# B&R Automation Studio project TD52 (part 3)

## Logical view

Binary libraries used (declarations not repeated): AsString, AsTime, BrSystem, DataObj, FileIO, LoopConR 2.72.0, LoopCont 3.03.1, Operator, Runtime, standard, SYS_LIB, CAN_Lib, AsXml, AsIecCon, AsArLog, AsIO, AsIODiag, AsIOAcc, AsARCfg, DRV_mbus, dvframe, AsTCP, AsArProf, AsNxDpS, AsNxPnS, ModDiag 1.10.1, AsBrMath, ArEventLog, AsBrStr, AsIOVib, AsFltGen, ArFirewall, AsHW, AsANSL, MpBackup 5.24.2, MpBase 5.24.1, SfDomain 5.24.1, AsEPL, MpJ1939 5.24.2, lSAFI_VCD

### Package Logical/Libraries - Global Libraries

### Library Logical/Libraries/AmmBase (IEC, version 4.13.0) - +
Depends on: standard

#### AmmBase.typ - Exported data types
```iecst
TYPE
	MM2AmmBase : 	STRUCT
		bGnlTrip1 : BOOL;
		bGnlTrip2 : BOOL;
		bGnlTrip3 : BOOL;
		bTriptype1 : BOOL;
		bTriptype2 : BOOL;
		bTriptype3 : BOOL;
		bGnlWarning : BOOL;
		iMsg : ARRAY[0..9999]OF USINT;
	END_STRUCT;
	AmmBase2MM : 	STRUCT
		bResetTrip : BOOL;
		bResetWarning : BOOL;
		bGnlTrip1 : BOOL;
		bGnlTrip2 : BOOL;
		bGnlTrip3 : BOOL;
		bGnlWarning : BOOL;
		bResetRiskClass0 : BOOL;
		bResetRiskClass1 : BOOL;
		bResetRiskClass2 : BOOL;
		bResetRiskClass3 : BOOL;
		bResetRiskClass4 : BOOL;
		iNumAlmTest : UDINT;
	END_STRUCT;
END_TYPE
```

#### AmmBase.fun - Exported functions and function blocks
```iecst
FUNCTION_BLOCK Msg (*AMM*)
	VAR_INPUT
		Num : UINT; (*alarm number*)
		Enable : BOOL; (*alarm enable*)
		Set : BOOL; (*alarm set*)
		PT : TIME; (*alarm delay*)
		Prio : UINT; (*alarm priority*)
		RiskClass : UINT; (*alarm riskclass*)
		Reset : BOOL; (*alarm reset*)
		LockReset : BOOL; (*alarm reset locked out*)
		AmmInAdr : UDINT;
		AmmOutAdr : UDINT;
	END_VAR
	VAR_OUTPUT
		Q : BOOL;
		Status : UINT;
		Test : BOOL; (*alarm test active*)
	END_VAR
	VAR
		xSR : SR;
		xTON : TON;
		bAlmTest : BOOL;
		MM2AB : REFERENCE TO MM2AmmBase;
		AB2MM : REFERENCE TO AmmBase2MM;
		bAdressErr : BOOL;
	END_VAR
	VAR CONSTANT
		FUB_Msg_InAdr_Err : UINT := 1111;
		FUB_Msg_OutAdr_Err : UINT := 2222;
	END_VAR
	VAR
		bRemoteReset : BOOL;
		AsArLogWrite_AMM : AsArLogWrite;
		AsArLogGetInfo_0 : AsArLogGetInfo;
		SetLog : BOOL;
		zzEdge00000 : BOOL;
	END_VAR
END_FUNCTION_BLOCK
```

- AmmBase.st (not readable text: treated as protected, skipped)

### Library Logical/Libraries/JEW_LIB1 (ANSIC, version 1.93.0)
Depends on: brsystem, SYS_LIB, brsystem, SYS_LIB

#### JEW_LIB1.fun
```iecst
FUNCTION_BLOCK FILTER
	VAR_INPUT
		In : INT;
		Filter : USINT;
		Reset : BOOL;
	END_VAR
	VAR_OUTPUT
		Out : INT;
	END_VAR
	VAR
		temp_mw : DINT;
	END_VAR
END_FUNCTION_BLOCK

FUNCTION_BLOCK FILTER_R
	VAR_INPUT
		In : REAL;
		Filter : UINT;
		Reset : BOOL;
	END_VAR
	VAR_OUTPUT
		Out : REAL;
	END_VAR
	VAR
		temp_mw : LREAL;
	END_VAR
END_FUNCTION_BLOCK

FUNCTION_BLOCK TimeBasedOnOff
	VAR_INPUT
		enable : BOOL;
		x : INT;
		min_value : INT;
		max_value : INT;
		tchange : UDINT;
		hysteresis : UINT;
		set_pos : INT;
		basetime : UDINT;
	END_VAR
	VAR_OUTPUT
		down : BOOL;
		up : BOOL;
		y : INT;
		status : UINT;
	END_VAR
	VAR
		y_act : REAL;
		fHystUp : REAL;
		fHystDown : REAL;
		fUnitTime : REAL;
		ulLastTime : UDINT;
		fDiffTime : REAL;
		fHysteresis : REAL;
	END_VAR
END_FUNCTION_BLOCK

FUNCTION_BLOCK TimeBasedOnOff_R
	VAR_INPUT
		enable : BOOL;
		x : REAL;
		min_value : REAL;
		max_value : REAL;
		tchange : REAL;
		hysteresis : REAL;
		set_pos : REAL;
		basetime : REAL;
	END_VAR
	VAR_OUTPUT
		down : BOOL;
		up : BOOL;
		y : REAL;
		status : UINT;
	END_VAR
	VAR
		y_act : REAL;
		fHystUp : REAL;
		fHystDown : REAL;
		fUnitTime : REAL;
		ulLastTime : REAL;
		fDiffTime : REAL;
		fHysteresis : REAL;
	END_VAR
END_FUNCTION_BLOCK

FUNCTION_BLOCK WDtoBIT
	VAR_INPUT
		Word : UINT;
	END_VAR
	VAR_OUTPUT
		Bit00 : BOOL;
		Bit01 : BOOL;
		Bit02 : BOOL;
		Bit03 : BOOL;
		Bit04 : BOOL;
		Bit05 : BOOL;
		Bit06 : BOOL;
		Bit07 : BOOL;
		Bit08 : BOOL;
		Bit09 : BOOL;
		Bit10 : BOOL;
		Bit11 : BOOL;
		Bit12 : BOOL;
		Bit13 : BOOL;
		Bit14 : BOOL;
		Bit15 : BOOL;
	END_VAR
END_FUNCTION_BLOCK

FUNCTION_BLOCK BITtoWD
	VAR_INPUT
		Bit00 : BOOL;
		Bit01 : BOOL;
		Bit02 : BOOL;
		Bit03 : BOOL;
		Bit04 : BOOL;
		Bit05 : BOOL;
		Bit06 : BOOL;
		Bit07 : BOOL;
		Bit08 : BOOL;
		Bit09 : BOOL;
		Bit10 : BOOL;
		Bit11 : BOOL;
		Bit12 : BOOL;
		Bit13 : BOOL;
		Bit14 : BOOL;
		Bit15 : BOOL;
	END_VAR
	VAR_OUTPUT
		Word : UINT;
	END_VAR
END_FUNCTION_BLOCK

FUNCTION_BLOCK PID_A
	VAR_INPUT
		enable : BOOL;
		init : BOOL;
		ist : INT;
		soll : INT;
		kp : INT;
		ki : INT;
		kd : INT;
		gunten : INT;
		goben : INT;
		C0 : DINT;
	END_VAR
	VAR_OUTPUT
		limit : BOOL;
		integr : DINT;
		stell : INT;
	END_VAR
	VAR
		ist_alt : INT;
	END_VAR
END_FUNCTION_BLOCK

FUNCTION_BLOCK PID_A_R
	VAR_INPUT
		enable : BOOL;
		init : BOOL;
		ist : REAL;
		soll : REAL;
		kp : INT;
		ki : INT;
		kd : INT;
		gunten : INT;
		goben : INT;
		C0 : DINT;
	END_VAR
	VAR_OUTPUT
		limit : BOOL;
		integr : DINT;
		stell : REAL;
	END_VAR
	VAR
		ist_alt : INT;
	END_VAR
END_FUNCTION_BLOCK

FUNCTION_BLOCK TON_R
	VAR_INPUT
		IN : BOOL;
		PT : UDINT;
		RS : BOOL;
	END_VAR
	VAR_OUTPUT
		Q : BOOL;
		ET : UDINT;
	END_VAR
	VAR
		init_old : USINT;
		tick_old : UDINT;
	END_VAR
END_FUNCTION_BLOCK

FUNCTION_BLOCK BH
	VAR_INPUT
		enable : BOOL;
		BH_adr : UDINT;
	END_VAR
	VAR_OUTPUT
		BH_Imp : BOOL;
		BM_Imp : BOOL;
	END_VAR
END_FUNCTION_BLOCK

FUNCTION_BLOCK RAMPE
	VAR_INPUT
		enable : BOOL;
		In : INT;
		Rise : UINT;
		Sink : UINT;
		TC_Time : UINT;
	END_VAR
	VAR_OUTPUT
		Out : INT;
	END_VAR
	VAR
		f_out : REAL;
	END_VAR
END_FUNCTION_BLOCK

FUNCTION_BLOCK RAMPE_R
	VAR_INPUT
		enable : BOOL;
		In : REAL;
		Rise : REAL;
		Sink : REAL;
		TC_Time : UINT;
	END_VAR
	VAR_OUTPUT
		Out : REAL;
	END_VAR
	VAR
		f_out : REAL;
	END_VAR
END_FUNCTION_BLOCK

FUNCTION_BLOCK GR_MIN_MAXR
	VAR_INPUT
		In : REAL;
		Gw : REAL;
		Hy_min : REAL;
		Hy_max : REAL;
	END_VAR
	VAR_OUTPUT
		Q : BOOL;
	END_VAR
END_FUNCTION_BLOCK

FUNCTION_BLOCK GR_MIN
	VAR_INPUT
		In : INT;
		Gw : INT;
		Hy : INT;
	END_VAR
	VAR_OUTPUT
		Q : BOOL;
	END_VAR
END_FUNCTION_BLOCK

FUNCTION_BLOCK GR_MINR
	VAR_INPUT
		In : REAL;
		Gw : REAL;
		Hy : REAL;
	END_VAR
	VAR_OUTPUT
		Q : BOOL;
	END_VAR
END_FUNCTION_BLOCK

FUNCTION us_BitClr : UINT
	VAR_INPUT
		In : UINT;
		BitNr : USINT;
	END_VAR
END_FUNCTION

FUNCTION_BLOCK GR_MAX
	VAR_INPUT
		In : INT;
		Gw : INT;
		Hy : INT;
	END_VAR
	VAR_OUTPUT
		Q : BOOL;
	END_VAR
END_FUNCTION_BLOCK

FUNCTION_BLOCK GR_MAXR
	VAR_INPUT
		In : REAL;
		Gw : REAL;
		Hy : REAL;
	END_VAR
	VAR_OUTPUT
		Q : BOOL;
	END_VAR
END_FUNCTION_BLOCK

FUNCTION us_BitSet : UINT
	VAR_INPUT
		In : UINT;
		BitNr : USINT;
	END_VAR
END_FUNCTION

FUNCTION us_BitTest : BOOL
	VAR_INPUT
		In : UINT;
		BitNr : USINT;
	END_VAR
END_FUNCTION

FUNCTION uc_BitClr : USINT
	VAR_INPUT
		In : USINT;
		BitNr : USINT;
	END_VAR
END_FUNCTION

FUNCTION uc_BitSet : USINT
	VAR_INPUT
		In : USINT;
		BitNr : USINT;
	END_VAR
END_FUNCTION

FUNCTION uc_BitTest : BOOL
	VAR_INPUT
		In : USINT;
		BitNr : USINT;
	END_VAR
END_FUNCTION

FUNCTION ul_BitSet : UDINT
	VAR_INPUT
		In : UDINT;
		BitNr : USINT;
	END_VAR
END_FUNCTION

FUNCTION ul_BitClr : UDINT
	VAR_INPUT
		In : UDINT;
		BitNr : USINT;
	END_VAR
END_FUNCTION

FUNCTION ul_BitTest : BOOL
	VAR_INPUT
		In : UDINT;
		BitNr : USINT;
	END_VAR
END_FUNCTION

FUNCTION ITOA : SINT
	VAR_INPUT
		In : INT;
		Out : STRING[7];
	END_VAR
END_FUNCTION

FUNCTION_BLOCK xSignScal
	VAR_INPUT
		enable : BOOL;
		num : UINT;
		param : UDINT;
		In : INT;
	END_VAR
	VAR_OUTPUT
		error : BOOL;
		exceed : BOOL;
		Out : INT;
	END_VAR
END_FUNCTION_BLOCK

FUNCTION_BLOCK xSignScal_R
	VAR_INPUT
		enable : BOOL;
		num : UINT;
		param : UDINT;
		In : REAL;
	END_VAR
	VAR_OUTPUT
		error : BOOL;
		exceed : BOOL;
		Out : REAL;
	END_VAR
END_FUNCTION_BLOCK

FUNCTION_BLOCK TOF_R
	VAR_INPUT
		IN : BOOL;
		PT : UDINT;
		RS : BOOL;
	END_VAR
	VAR_OUTPUT
		Q : BOOL;
		ET : UDINT;
	END_VAR
	VAR
		init_old : UDINT;
		tick_old : UDINT;
	END_VAR
END_FUNCTION_BLOCK

FUNCTION_BLOCK TP_R
	VAR_INPUT
		IN : BOOL;
		PT : UDINT;
		RS : BOOL;
	END_VAR
	VAR_OUTPUT
		Q : BOOL;
		ET : UDINT;
	END_VAR
	VAR
		init_old : USINT;
		tick_old : UDINT;
		IN_old : BOOL;
	END_VAR
END_FUNCTION_BLOCK
```

#### JEW_LIB1.typ
```iecst
TYPE
	bh_typ : STRUCT
		tick	: USINT ;
		second	: USINT ;
		minute	: USINT ;
		spare	: USINT ;
	END_STRUCT;
END_TYPE
```

#### bh.c
```c
/***********************************************************************************
* Name      : bh.c
* Titel     : Betriebsstundengenerierung
* Version   : V1.10
* Datum     : 17.05.2002
*
* Uebergabe : enable			BOOL			Betriebsstundengenerierung aus/ein
*
* Rueckgabe : BH_adr	 struct USINT tick		Sekundentakt
*							    USINT second	Sekundenzaehler
*							    USINT minute	Minutenzähler
*								USINT spare		Reserve
*			  BH_Imp			BOOL			Betriebsstundenimpuls
*
* History   :
*  V1.00	  14.09.1998,fw			erstellt
*  V1.01	  24.08.2001,Fa.		fd->BD_adr durch fd->BH_adr ersetzt
*  V1.10	  17.05.2002,fw			#include <burtrap.h> durch <sys_lib.h> ersetzt
*  V1.70	  17.06.2002,WeitzerT	inc. plctypes entf.; bei jewlib1.h <> statt ""
*  V1.70.1	  24.01.2014,WeitzerT	correction of compiler warnings
*  V1.93.0	  27.10.2023,Zuschnig	Include minute impuls
*
***********************************************************************************/
#include <jew_lib1.h>
#include <sys_lib.h>

void BH(BH_typ *fd)
{
	UINT	ticks;
	bh_typ	*bh_adr;

	bh_adr = (bh_typ*)fd->BH_adr;

	fd->BH_Imp = 0;							/* vorab Stundenimpuls reset */
	fd->BM_Imp = 0;							/* vorab Minutenimpuls reset */

	if (fd->enable == 1)
	{
		ticks = 0;							/* Zwischenzeitlich für Änderung auf i386 */

		ticks = TIM_ticks();				/* 10 ms Takt auslesen */

		if ((ticks < 50) && (bh_adr->tick == 0))
		{
			bh_adr->tick = 1;				/* Sekundentakt setzen */
			++bh_adr->second;				/* im Sekundentakt zaehlen */
			if (bh_adr->second > 59)
			{
				bh_adr->second = 0;
				fd->BM_Imp = 1;				/* Minutenimpuls ausgeben */
				++bh_adr->minute;			/* im Minutetakt zaehlen */
				if (bh_adr->minute > 59)
				{
					fd->BH_Imp = 1;			/* Stundenimpuls ausgeben */
					bh_adr->minute = 0;
				}
			}
		}
		else if ((ticks > 50) && (bh_adr->tick == 1))
			bh_adr->tick = 0;				/* Sekundentakt ruecksetzen */
	}
}
```

#### bittowd.c
```c
/***********************************************************************************
* Name      : BITtoWD.c
* Titel     : 16 Bits auf ein Word(2Byte) komprimieren
* Version   : V1.00
* Datum     : 09.11.1998
*
* Uebergabe : Bit00		BOOL	Bit 00 des Ausgangswortes
*			  Bit01		BOOL	Bit 01 des Ausgangswortes
*			  Bit02		BOOL	Bit 02 des Ausgangswortes
*			  Bit03		BOOL	Bit 03 des Ausgangswortes
*			  Bit04		BOOL	Bit 04 des Ausgangswortes
*			  Bit05		BOOL	Bit 05 des Ausgangswortes
*			  Bit06		BOOL	Bit 06 des Ausgangswortes
*			  Bit07		BOOL	Bit 07 des Ausgangswortes
*			  Bit08		BOOL	Bit 08 des Ausgangswortes
*			  Bit09		BOOL	Bit 09 des Ausgangswortes
*			  Bit10		BOOL	Bit 10 des Ausgangswortes
*			  Bit11		BOOL	Bit 11 des Ausgangswortes
*			  Bit12		BOOL	Bit 12 des Ausgangswortes
*			  Bit13		BOOL	Bit 13 des Ausgangswortes
*			  Bit14		BOOL	Bit 14 des Ausgangswortes
*			  Bit15		BOOL	Bit 15 des Ausgangswortes
*
* Rueckgabe : Word 		UINT	Kompriemiertes Eingangsabbild
*
* History   :
*  V1.00	  09.11.1998,fw			erstellt
*  V1.70	  17.06.2002,WeitzerT	inc. plctypes entf.; bei jewlib1.h <> statt ""
*
***********************************************************************************/
#include <jew_lib1.h>

void BITtoWD(BITtoWD_typ *fd)
{
	fd->Word = fd->Bit15;
	fd->Word = ((fd->Word)<<1) + fd->Bit14;
	fd->Word = ((fd->Word)<<1) + fd->Bit13;
	fd->Word = ((fd->Word)<<1) + fd->Bit12;
	fd->Word = ((fd->Word)<<1) + fd->Bit11;
	fd->Word = ((fd->Word)<<1) + fd->Bit10;
	fd->Word = ((fd->Word)<<1) + fd->Bit09;
	fd->Word = ((fd->Word)<<1) + fd->Bit08;
	fd->Word = ((fd->Word)<<1) + fd->Bit07;
	fd->Word = ((fd->Word)<<1) + fd->Bit06;
	fd->Word = ((fd->Word)<<1) + fd->Bit05;
	fd->Word = ((fd->Word)<<1) + fd->Bit04;
	fd->Word = ((fd->Word)<<1) + fd->Bit03;
	fd->Word = ((fd->Word)<<1) + fd->Bit02;
	fd->Word = ((fd->Word)<<1) + fd->Bit01;
	fd->Word = ((fd->Word)<<1) + fd->Bit00;
}
```

#### filter.c
```c
/***********************************************************************************
* Name      : filter.c
* Titel     : Filter mit PT1-Verhalten
* Version   : V1.0
* Datum     : 14.09.1998
*
* Uebergabe : In		INT		Eingangssignal
*			  Filter	SINT	Filterkonstante filter = T1 / T (T1 = Verzoegerung 1. Ordnung)
*
* Rueckgabe : Out	 	INT		Ausgangssignal
*
* History   :
*  V1.00	  14.09.1998,fw		erstellt
*  V1.20      21.12.1998,BK		Zeitkonstante im .h-File von SINT auf USINT
*  V1.70	  17.06.2002,WeitzerT	inc. plctypes entf.; bei jewlib1.h <> statt ""
*  V1.91	  02.02.2022,Schmid		added Reset input
*
***********************************************************************************/
#include <jew_lib1.h>

void FILTER(FILTER_typ *fd)
{
	if (fd->Filter == 0)
		fd->Filter = 1;				/* Division durch 0 verhindern */

	if (fd->Reset)
		fd->temp_mw = fd->In * fd->Filter;
	else
		fd->temp_mw = fd->temp_mw + fd->In - fd->Out;

	fd->Out = (int)(fd->temp_mw/fd->Filter);
}
```

#### gr_max.c
```c
/***********************************************************************************
* Name      : gr_max.c
* Titel     : Maximal-Grenzwertkontrolle mit Hysterese
* Version   : V1.3
* Datum     : 28.09.1999
*
* Uebergabe : In		INT		Eingangssignal
*			  Gw		INT		Grenzwert
*			  Hy		INT		Hysterese
*
* Rueckgabe : Q	 		INT		Ausgangssignal = 1 => Grenzwert ueberschritten
*
* History   :
*  V1.00	  14.09.1998,fw			erstellt
*  V1.30      28.09.1999,BrunnerK	Vergleichsoperanden wurden geaendert
*  V1.70	  17.06.2002,WeitzerT	inc. plctypes entf.; bei jewlib1.h <> statt ""
*
***********************************************************************************/
#include <jew_lib1.h>

void GR_MAX(GR_MAX_typ *fd)
{
	if (fd->In >= fd->Gw)
		fd->Q = 1;
	else if (fd->In < (fd->Gw - fd->Hy))
		fd->Q = 0;
}
```

#### gr_min_maxR.c
```c
/***********************************************************************************
* Name      : gr_min_max.c
* Titel     : Maximal- and Minimum Grenzwertkontrolle mit Hysterese
* Version   : V1.3
* Datum     : 26.05.2015
*
* Uebergabe : In		INT		Eingangssignal
*			  Gw		INT		Grenzwert
*			  Hy_min	INT		Hysterese - Down limit
*			  Hy_max	INT		Hysterese - Up Limit
*
* Rueckgabe : Q	 		INT		Ausgangssignal = 1 => Grenzwert ueberschritten
*
* History   :
*  V1.00	  28.05.2015,Walid Mari  Erstellt, basiert auf GR_MAXR library
*
***********************************************************************************/
#include <jew_lib1.h>

void GR_MIN_MAXR(GR_MIN_MAXR_typ *fd)
{
	if 		(fd->In >=( fd->Gw	+	fd->Hy_max))
		fd->Q = 1;
	else if (fd->In < (fd->Gw 	- 	fd->Hy_min))
		fd->Q = 0;
}
```

#### gr_maxR.c
```c
/***********************************************************************************
* Name      : gr_max.c
* Titel     : Maximal-Grenzwertkontrolle mit Hysterese
* Version   : V1.3
* Datum     : 28.09.1999
*
* Uebergabe : In		INT		Eingangssignal
*			  Gw		INT		Grenzwert
*			  Hy		INT		Hysterese
*
* Rueckgabe : Q	 		INT		Ausgangssignal = 1 => Grenzwert ueberschritten
*
* History   :
*  V1.00	  14.09.1998,fw			erstellt
*  V1.30      28.09.1999,BrunnerK	Vergleichsoperanden wurden geaendert
*  V1.70	  17.06.2002,WeitzerT	inc. plctypes entf.; bei jewlib1.h <> statt ""
*
***********************************************************************************/
#include <jew_lib1.h>

void GR_MAXR(GR_MAXR_typ *fd)
{
	if (fd->In >= fd->Gw)
		fd->Q = 1;
	else if (fd->In < (fd->Gw - fd->Hy))
		fd->Q = 0;
}
```

#### gr_min.c
```c
/***********************************************************************************
* Name      : gr_min.c
* Titel     : Minimal-Grenzwertkontrolle mit Hysterese
* Version   : V1.3
* Datum     : 28.09.1999
*
* Uebergabe : In		INT		Eingangssignal
*			  Gw		INT		Grenzwert
*			  Hy		INT		Hysterese
*
* Rueckgabe : Q	 		INT		Ausgangssignal = 1 => Grenzwert unterschritten
*
* History   :
*  V1.00	  14.09.1998,fw			erstellt
*  V1.30      28.09.1999,BrunnerK	Vergleichsoperanden wurden geaendert
*  V1.70	  17.06.2002,WeitzerT	inc. plctypes entf.; bei jewlib1.h <> statt ""
*
***********************************************************************************/
#include <jew_lib1.h>

void GR_MIN(GR_MIN_typ *fd)
{
	if (fd->In <= fd->Gw)
		fd->Q = 1;
	else if (fd->In > (fd->Gw + fd->Hy))
		fd->Q = 0;
}
```

#### itoa.c
```c
/***********************************************************************************
* Name      : itoa.c
* Titel     : Konvertierung Integer to ASCII-String
* Version   : V1.3
* Datum     : 30.09.1999
*
* Uebergabe : Strukturvariable:
*             In		INT		Zu konvertierender Integerwert
*			  *pCharFld	SINT	Pointer auf das Char-Array
*
* Rueckgabe : Strukturvariable:
*			  StrLen	SINT	Laenge des Strings
*
* History   :
*  V1.00	  xx.xx.1998,fw			erstellt
*  V1.30      30.09.1999,BrunnerK	In Library umgewandelt
*  V1.70	  17.06.2002,WeitzerT	inc. plctypes entf.; bei jewlib1.h <> statt ""
*  V1.70.1	  24.01.2014,WeitzerT	correction of compiler warnings
*
***********************************************************************************/
#include <jew_lib1.h>

signed char ITOA(signed short In, plcstring* Out)

{
	signed short	i, string_len, neg;
	signed long		val;
	signed short	InTemp;

	string_len = 1;					/* minimum 1 Zeichen lang */
	neg = 0;						/* vorab Wert positiv */
	InTemp = 0;

	if (In<0)
	{								/* Wert negativ */
		InTemp = In;				/* Negative Wert sichern */
/*		In = abs(In);				   Absolutbetrag bilden */
		neg = 1;					/* Kennung Wert ist negativ setzen */
		string_len++;				/* String wird um das Vorzeichen länger */
		Out[0] = '-';		    	/* Vorzeichen am Stringanfang eintragen */
	}

	val = In;
	while((val= val/10) != 0)		/* Berechnung der Stringlänge */
	{
		string_len++;
	}

	val = In;
	Out[string_len] = 0;		/* Stringendekennung eintragen */

	for(i=0; i<(string_len-neg); ++i)	/* Wert ASCII wandeln */
	{
		Out[string_len-i-1] = (char)((val % 10) + '0');
		val = val / 10;
	}

	if (neg == 1)
	{
		In = InTemp;				/* Negativen Wert zuruecksichern */
	}

	return string_len;				/* Stringlänge ohne Stringendekennung */
}
```

#### pid_a_R.c
```c
/********************************************************************
 * COPYRIGHT -- INNIO Company
 ********************************************************************
 * Library: JEW_LIB1
 * File: pid_a_R.c
 * Author: 320003156
 * Created: August 17, 2011
 * Modified: 2017-08-08 FW   adapted for GCC 4.1.2.
 *******************************************************************/

#include <bur/plc.h>
#include <JEW_LIB1.h>

void PID_A_R(PID_A_R_typ* pida)
{
	/* Deklaration Zwischenablage */
	long	stell_neu;
	short	e;

	if (pida->enable)
	{
		/* Initialisierung Regler */
		if (pida->init)
		{
			pida->integr = pida->C0;
			pida->ist_alt = 0;
		}

		/* Rücksetzen von Limitfehler */
		pida->limit = 0;

		/* Regler - Algorythmus
		yi = yi_1 + (e + ist_alt)/2 * ki
		stell  = (yp + yi + yd) / 256
		stell  = (e*kp + yi + (ist_alt - e) * (kd * -1)) / 256
		*/

		/* Berechnung Regelabweichung */
		e = pida->soll - pida->ist;

		/* Berechnung Integralanteil */
		pida->integr = pida->integr + (pida->ki) * ((e + pida->ist_alt) >> 1);

		/* Berechnung Stellgröße */
		stell_neu = (pida->kp * e + pida->integr - pida->kd * (pida->ist_alt - e)) >> 8;

		/* Übergabe an Schnittstelle */
	    pida->stell = stell_neu;

		/* Prüfung und Begrenzung des Stellsignales */
        if (stell_neu < pida->gunten)
		{
			pida->limit = 1;
			if (pida->ki != 0) pida->integr = (pida->gunten << 8) - (pida->kp * e - pida->kd * (e - pida->ist_alt));
			pida->stell = pida->gunten;
		}
		else if (stell_neu > pida->goben)
		{
			pida->limit = 1;
			if (pida->ki != 0) pida->integr = (pida->goben << 8) - (pida->kp * e - pida->kd * (e - pida->ist_alt));
			pida->stell = pida->goben;
		}

		/* Übergabe für neue Berechnug */
		pida->ist_alt = e;

	}
}
```

#### pid_a.c
```c
/************************************************************************************
* Name      : pid_a.src                                                         	*
* Titel     : Einfacher PID-Regler auf Integer-Basis                               	*
*												                            	   	*
* Uebergabe : enable	BOOL	Freigabe											*
*			  init		BOOL	Initialisierung									   	*
*			  ist		INT		Inputvariablen, Istwert                         	*
*			  soll		INT		Sollwert                            	  			*
*			  kp		INT		Proportionalverstärkung                             *
*			  ki		INT		Integrationsbeiwert                                 *
*			  kd		INT		Differenzierbeiwert                                 *
*			  gunten	INT		unterer Grenzwert                              	   	*
*			  goben		INT		oberer Grenzwert                            	   	*
*			  C0		DINT	Integrator Startwert wird übernommen wenn !=0	   	*
*												                            	   	*
* Rueckgabe : limit		BOOL	Limit Stellgrenzwert unter-/Überschritten			*
*			  integr	DINT	Integrator              							*
*			  stell		INT		Outputvariable, Stellwert                           *
*												                       				*
* Lok. Var. : e			INT		Reglelabweichung aktuell							*
*			  ist_alt		INT		alte Regelabweichung für Differenzbildung			*
*			  stell_neu DINT	Zwischenspeicherung des Stellwertes					*
*												                            	   	*
* History   :	                            	   								   	*
* V1.00	  	  06.06.2002,tw		erstellt										   	*
* V1.10       2017-08-08 FW   adapted for GCC 4.1.2.
*																				   	*
*************************************************************************************
*               		                                                           	*
*  BESCHREIBUNG:        		                                                   	*
*  -------------                		                                           	*
*                                       		                                   	*
*  Der FUB PID_a realisiert einen einfachen PID-Algorithmus, der auf		       	*
*  unterschreiten der unteren Stellwertgrenze <gunten> und auf             		   	*
*  überschreiten der oberen Stellwertgrenze <goben> überwacht. In diesem		   	*
*  Fall wird der Integrator neu berechnet und der Stellwert gemäß der     		   	*
*  Grenze begrenzt.                                                       		   	*
*  Der Integrator <integr> muß beim erstmaligen Aufruf des FUB richtig    		   	*
*  initialisiert werden (in der Regel mit 0).                             		   	*
*  Die Regelparameter der FUB-Schnittstelle sind wegen der Integerrechnung		   	*
*  mit 256 zu multiplizieren, das untere Byte entspricht demnach der Stelle		   	*
*  hinter dem Komma.                                                      		   	*
*                                                                         		   	*
************************************************************************************/
#include <bur/plc.h>
#include <JEW_LIB1.h>

void PID_A(PID_A_typ* pida)
{
	/* Deklaration Zwischenablage */
	long	stell_neu;
	short	e;

	if (pida->enable)
	{
		/* Initialisierung Regler */
		if (pida->init)
		{
			pida->integr = pida->C0;
			pida->ist_alt = 0;
		}

		/* Rücksetzen von Limitfehler */
		pida->limit = 0;

		/* Regler - Algorythmus
		yi = yi_1 + (e + ist_alt)/2 * ki
		stell  = (yp + yi + yd) / 256
		stell  = (e*kp + yi + (ist_alt - e) * (kd * -1)) / 256
		*/

		/* Berechnung Regelabweichung */
		e = pida->soll - pida->ist;

		/* Berechnung Integralanteil */
		pida->integr = pida->integr + (pida->ki) * ((e + pida->ist_alt) >> 1);

		/* Berechnung Stellgröße */
		stell_neu = (pida->kp * e + pida->integr - pida->kd * (pida->ist_alt - e)) >> 8;

		/* Übergabe an Schnittstelle */
	    pida->stell = stell_neu;

		/* Prüfung und Begrenzung des Stellsignales */
        if (stell_neu < pida->gunten)
		{
			pida->limit = 1;
			if (pida->ki != 0) pida->integr = (pida->gunten << 8) - (pida->kp * e - pida->kd * (e - pida->ist_alt));
			pida->stell = pida->gunten;
		}
		else if (stell_neu > pida->goben)
		{
			pida->limit = 1;
			if (pida->ki != 0) pida->integr = (pida->goben << 8) - (pida->kp * e - pida->kd * (e - pida->ist_alt));
			pida->stell = pida->goben;
		}

		/* Übergabe für neue Berechnug */
		pida->ist_alt = e;

	}
}
```

#### rampe_R.c
```c
/********************************************************************
 * COPYRIGHT -- INNIO Company
 ********************************************************************
 * Library: JEW_LIB1
 * File: rampe_R.c
 * Author: 320003156
 * Created: August 17, 2011
 *******************************************************************/

#include <jew_lib1.h>

void RAMPE_R(RAMPE_R_typ *fd)
{
	if (fd->enable)
	{
		if (fd->Out < fd->In)
		{
			fd->f_out = fd->f_out + (0.001 * fd->Rise * fd->TC_Time);
			if (fd->f_out > fd->In)
				fd->f_out = fd->In;
		}
		else if (fd->Out > fd->In)
		{
			fd->f_out = fd->f_out - (0.001 * fd->Sink * fd->TC_Time);
			if (fd->f_out < fd->In)
				fd->f_out = fd->In;
		}

		fd->Out = fd->f_out;
	}
	else
	{
		fd->Out = fd->In;
		fd->f_out = fd->In;
	}
}
```

#### us_bitset.c
```c
/***********************************************************************************
* Name      : us_BitSet.c
* Titel     : Setzen einer Bit-Stelle eines unsigned short auf TRUE
* Version   : V1.0
* Datum     : 15.10.2001
*
* Uebergabe : In				UINT			Wert mit zu setzender Bit Stelle
*			: BitNr				USINT			Bit Stelle die gesetzt werden soll
*
* Rueckgabe : function			UINT			Wert mit gesetzter Bit Stelle
*
* History   :
*  V1.00	  15.10.2001,Fa			erstellt
*  V1.70	  17.06.2002,WeitzerT	bei jewlib1.h <> statt ""
*
***********************************************************************************/
#include <jew_lib1.h>

unsigned short us_BitSet(unsigned short In, unsigned char BitNr)
{
	return  ( In | (1 << BitNr));
}
```

#### rampe.c
```c
/***********************************************************************************
* Name      : rampe.c
* Titel     : Rampengenerierung
* Version   : V1.0
* Datum     : 14.09.1998
*
* Uebergabe : enable	BOOL	Freigabe 0 => Out = in / 1 => Out = rampe(in)
*			  In		INT		Eingangssignal
*			  Rise		UINT	positive Aenderung / s
*			  Sink		UINT	negative Aenderung / s
*			  TC_Time	UINT	Zykluszeit der Taskklasse in [ms]
*
* Rueckgabe : Out	 	INT		Ausgangssignal
*
* History   :
*  V1.00	  14.09.1998,fw			erstellt
*  V1.70	  17.06.2002,WeitzerT	inc. plctypes entf.; bei jewlib1.h <> statt ""
*
***********************************************************************************/
#include <jew_lib1.h>

void RAMPE(RAMPE_typ *fd)
{
	if (fd->enable)
	{
		if (fd->Out < fd->In)
		{
			fd->f_out = fd->f_out + (0.001 * fd->Rise * fd->TC_Time);
			if (fd->f_out > fd->In)
				fd->f_out = fd->In;
		}
		else if (fd->Out > fd->In)
		{
			fd->f_out = fd->f_out - (0.001 * fd->Sink * fd->TC_Time);
			if (fd->f_out < fd->In)
				fd->f_out = fd->In;
		}

		fd->Out = (short int)(fd->f_out);
	}
	else
	{
		fd->Out = fd->In;
		fd->f_out = fd->In;
	}
}
```

#### timebasedonoff_R.c
```c
/********************************************************************
 * COPYRIGHT -- INNIO Company
 ********************************************************************
 * Library: JEW_LIB1
 * File: timebasedonoff_R.c
 * Author: 320003156
 * Created: August 23, 2011
 *******************************************************************/

#include <jew_lib1.h>
#include <bur/plctypes.h>

void TimeBasedOnOff(TimeBasedOnOff_typ *fd)
/* begin FUB */
{

if (fd->enable != 0)
{
	fd->status = 0;		/* reset status */

	/* calculate basetime for 1 step of x */
	if (fd->tchange != 0)
	{
		fd->fUnitTime = (float)(fd->max_value - fd->min_value)/fd->tchange;
	}
	else
	{
		fd->status = 1;		/* no change time from min_value to max_value */
	}

	/* calcualte time difference since last cycle */
	fd->fDiffTime = fd->basetime - fd->ulLastTime;

	/* calculate minimum hysteresis for the next step */
	fd->fHysteresis = fd->fUnitTime*fd->fDiffTime;

	/* calculate actual position and hysteresis for the next step */
	if (fd->up != 0) 	/* open actuator */
	{
		fd->y_act   = fd->y_act + fd->fHysteresis;		/* calcualte new actual position = y_act + fDiffTime*fUnitTime*/

		fd->fHystUp = fd->fHysteresis;					/* set to minimum up hystersis */

		if (fd->fHysteresis < fd->hysteresis)		/* is mimimum hysteresis < user hysteresis */
		{
			fd->fHystDown = fd->hysteresis;		/* use user down hysteresis */
		}
		else
		{
			fd->fHystDown = fd->fHysteresis;	/* set to minimum down hysteresis */
		}

	}
	else if (fd->down != 0)		/* close actuator */
	{
		fd->y_act     = fd->y_act - fd->fHysteresis;		/* calcualte new actual position close = y_act - fDiffTime*fUnitTime*/

		fd->fHystDown = fd->fHysteresis;					/* set to minimum down hysteresis */

		if (fd->fHysteresis < fd->hysteresis)		/* is mimimum hysteresis < user hysteresis */
		{
			fd->fHystUp = fd->hysteresis;		/* use user up hysteresis */
		}
		else
		{
			fd->fHystUp = fd->fHysteresis;		/* set to minimum up hysteresis */
		}
	}
	else		/* actuator stopped */
	{
		if (fd->fHysteresis < fd->hysteresis)		/* is mimimum hysteresis < user hysteresis */
		{
			fd->fHystUp   = fd->hysteresis;		/* use user up hysteresis */
			fd->fHystDown = fd->fHystUp;		/* use user down hysteresis */
		}
		else
		{
			fd->fHystUp   = fd->fHysteresis;		/* set to minimum up hysteresis */
			fd->fHystDown = fd->fHystUp;			/* set to minimum down hysteresis */
		}
	}

	if (fd->x >= fd->y_act + fd->fHystUp)		/* setpoint position >= actual position + hysteresis */
	{
		fd->up   = 1;		/* set bit for open */
		fd->down = 0;		/* reset bit for close */
	}
	else if (fd->x <= fd->y_act - fd->fHystDown)		/* setpoint position <= actual position - hysteresis */
	{
		fd->down = 1;		/* set bit for close */
		fd->up   = 0;		/* reset bit for open */
	}
	else		/* if difference between actual and setpoint positioin within hystetrsis */
	{
		fd->up   = 0;		/* reset bit for open */
		fd->down = 0;		/* reset bit for close */
	}
}
else
{
	fd->y_act = fd->set_pos;
}

if (fd->y_act >= 0)	/* check pos. or neg. output and compensate rounding error */
{
	fd->y          = (fd->y_act+0.5);	/* actual position FUB output */
}
else
{
	fd->y          = (fd->y_act-0.5);	/* actual position FUB output */
}

fd->ulLastTime = fd->basetime;				/* save last cycle time */

/* end FUB */
}
```

#### timebasedonoff.c
```c
/*******************************************************************************
JEW_LIB1: time based on/off in dependence of setpoint an actual position
Copyright 1998 - 2003 Jenbacher AG

- calculate actual position and hysteresis for the next step
- output actual position

Customized modifications:
------------------------

History:
-------
V0.1	02-11-2002	Weitzer,	generated from TimeBaseOn.SRC / V0.1 / 02-11-2002 /Fahringer
V0.2	28-03-2003	Fahringer,	correct casting for calculation of	fd->fUnitTime

Instructions for use:
--------------------
enable	   	FUB on / off
x			setpoint position
min_value  	min position
max_value  	maximum positon
hysteresis  minimum difference between x and y_act for drive to new position
tchange    	time for drive from min_value to max_value
basetime   	time base for FUB timing  (best generated by LCCounter FUB)
status		FUB status 0 = OK, 1 = no difference between max_value and min_value
up			open actuator
down		close actuator
y_act		actual actuator position (calcualted FUB internal)
set_pos		position if FUB is disabled (enable OFF)

Outstandings:
------------
*******************************************************************************/

#include <jew_lib1.h>
#include <bur/plctypes.h>

void TimeBasedOnOff_R(TimeBasedOnOff_R_typ *fd)
/* begin FUB */
{

if (fd->enable != 0)
{
	fd->status = 0;		/* reset status */

	/* calculate basetime for 1 step of x */
	if (fd->tchange != 0)
	{
		fd->fUnitTime = (float)(fd->max_value - fd->min_value)/fd->tchange;
	}
	else
	{
		fd->status = 1;		/* no change time from min_value to max_value */
	}

	/* calcualte time difference since last cycle */
	fd->fDiffTime = fd->basetime - fd->ulLastTime;

	/* calculate minimum hysteresis for the next step */
	fd->fHysteresis = fd->fUnitTime*fd->fDiffTime;

	/* calculate actual position and hysteresis for the next step */
	if (fd->up != 0) 	/* open actuator */
	{
		fd->y_act   = fd->y_act + fd->fHysteresis;		/* calcualte new actual position = y_act + fDiffTime*fUnitTime*/

		fd->fHystUp = fd->fHysteresis;					/* set to minimum up hystersis */

		if (fd->fHysteresis < fd->hysteresis)		/* is mimimum hysteresis < user hysteresis */
		{
			fd->fHystDown = fd->hysteresis;		/* use user down hysteresis */
		}
		else
		{
			fd->fHystDown = fd->fHysteresis;	/* set to minimum down hysteresis */
		}

	}
	else if (fd->down != 0)		/* close actuator */
	{
		fd->y_act     = fd->y_act - fd->fHysteresis;		/* calcualte new actual position close = y_act - fDiffTime*fUnitTime*/

		fd->fHystDown = fd->fHysteresis;					/* set to minimum down hysteresis */

		if (fd->fHysteresis < fd->hysteresis)		/* is mimimum hysteresis < user hysteresis */
		{
			fd->fHystUp = fd->hysteresis;		/* use user up hysteresis */
		}
		else
		{
			fd->fHystUp = fd->fHysteresis;		/* set to minimum up hysteresis */
		}
	}
	else		/* actuator stopped */
	{
		if (fd->fHysteresis < fd->hysteresis)		/* is mimimum hysteresis < user hysteresis */
		{
			fd->fHystUp   = fd->hysteresis;		/* use user up hysteresis */
			fd->fHystDown = fd->fHystUp;		/* use user down hysteresis */
		}
		else
		{
			fd->fHystUp   = fd->fHysteresis;		/* set to minimum up hysteresis */
			fd->fHystDown = fd->fHystUp;			/* set to minimum down hysteresis */
		}
	}

	if (fd->x >= fd->y_act + fd->fHystUp)		/* setpoint position >= actual position + hysteresis */
	{
		fd->up   = 1;		/* set bit for open */
		fd->down = 0;		/* reset bit for close */
	}
	else if (fd->x <= fd->y_act - fd->fHystDown)		/* setpoint position <= actual position - hysteresis */
	{
		fd->down = 1;		/* set bit for close */
		fd->up   = 0;		/* reset bit for open */
	}
	else		/* if difference between actual and setpoint positioin within hystetrsis */
	{
		fd->up   = 0;		/* reset bit for open */
		fd->down = 0;		/* reset bit for close */
	}
}
else
{
	fd->y_act = fd->set_pos;
}

if (fd->y_act >= 0)	/* check pos. or neg. output and compensate rounding error */
{
	fd->y          = (short)(fd->y_act+0.5);	/* actual position FUB output */
}
else
{
	fd->y          = (short)(fd->y_act-0.5);	/* actual position FUB output */
}

fd->ulLastTime = fd->basetime;				/* save last cycle time */

/* end FUB */
}
```

#### tof_r.c
```c
/***********************************************************************************
* Name      : tof_r.c
* Titel     : Abfallverzoegerung mit Reset-Eingang
* Version   : V1.10
* Datum     : 17.05.2002
*
* Uebergabe : IN		BOOL	Eingangssignal
*			  PT		UDINT	gewuenschte Verzoegerungszeit in [10 ms]
*			  RS		BOOL	Reseteingang: Durch Setzen dieses Eingangs wird der Ausgang Q sofort rueckgesetzt.
*
* Rueckgabe : Q	 		BOOL	Ausgangssignal
*			  PT		UDINT	abgelaufene Verzoegerungszeit in [10 ms]
*
* History   :
*  V1.00	  14.09.1998,fw			erstellt
*  V1.10      17.05.2002,fw     	Funktion SYS_info durch Funtionsblock SysInfo ersetzt,
*                               	damit die Library auch für i386 kompiliert werden kann.
*  V1.70	  17.06.2002,WeitzerT	inc. plctypes entf.; bei jewlib1.h <> statt ""
*
***********************************************************************************/
#include <jew_lib1.h>
#include <brsystem.h>

void TOF_R(TOF_R_typ *fd)
{
	SysInfo_typ	SysInf;
	unsigned long time_over;

	SysInf.enable = 1;
	SysInfo(&SysInf);

	if (fd->IN == 1)
		fd->Q = 1;

	if ((fd->IN == 0) && (fd->Q == 1))
	{
		if (SysInf.tick_count >= fd->tick_old)
			time_over = SysInf.tick_count - fd->tick_old;
		else
			time_over = 0 - fd->tick_old + SysInf.tick_count;

		fd->ET = fd->ET + time_over;

		if (fd->ET >= fd->PT)
		{
			fd->Q = 0;
			fd->ET = 0;
		}

		if (SysInf.init_count != fd->init_old)
		{
			fd->ET = 0;
			fd->init_old = SysInf.init_count;
		}
	}

	if (fd->RS == 1)
	{
		fd->Q = 0;
		fd->ET = 0;
	}

	fd->tick_old = SysInf.tick_count;

}
```

#### ton_r.c
```c
/***********************************************************************************
* Name      : ton_r.c
* Titel     : Anzugsverzoegerung mit Reset-Eingang
* Version   : V1.10
* Datum     : 17.05.2002
*
* Uebergabe : IN		BOOL	Eingangssignal
*			  PT		UDINT	gewuenschte Verzoegerungszeit in [10 ms]
*			  RS		BOOL	Reseteingang: Durch Setzen dieses Eingangs wird der Ausgang Q sofort rueckgesetzt.
*
* Rueckgabe : Q	 		BOOL	Ausgangssignal
*			  PT		UDINT	abgelaufene Verzoegerungszeit in [10 ms]
*
* History   :
*  V1.00	  14.09.1998,fw			erstellt
*  V1.10      17.05.2002,fw    		Funktion SYS_info durch Funktionsblock SysInfo ersetzt,
*                           	    damit die Libary auch für i386 kompiliert werden kann.
*  V1.70	  17.06.2002,WeitzerT	inc. plctypes entf.; bei jewlib1.h <> statt ""
*
***********************************************************************************/
#include <jew_lib1.h>
#include <brsystem.h>

void TON_R(TON_R_typ *fd)
{
	SysInfo_typ	SysInf;
	unsigned long time_over;

	SysInf.enable = 1;
	SysInfo(&SysInf);

	if (fd->IN == 1)
	{
		if (SysInf.tick_count >= fd->tick_old)
			time_over = SysInf.tick_count - fd->tick_old;
		else
			time_over = 0 - fd->tick_old + SysInf.tick_count;

		fd->ET = fd->ET + time_over;

		if (fd->ET >= fd->PT)
		{
			fd->Q = 1;
			fd->ET = fd->PT;
		}

		if (SysInf.init_count != fd->init_old)
		{
			fd->Q = 0;
			fd->ET = 0;
			fd->init_old = SysInf.init_count;
		}
	}
	else
	{
		fd->Q = 0;
		fd->ET = 0;
	}

	if (fd->RS == 1)
	{
		fd->Q = 0;
		fd->ET = 0;
	}

	fd->tick_old = SysInf.tick_count;

}
```

#### tp_r.c
```c
/***********************************************************************************
* Name      : tp_r.c
* Titel     : Pulsgenerierung Reset-Eingang
* Version   : V1.10
* Datum     : 17.05.2002
*
* Uebergabe : IN		BOOL	Eingangssignal
*			  PT		UDINT	gewuenschte Pulsdauer in [10 ms]
*			  RS		BOOL	Reseteingang: Durch Setzen dieses Eingangs wird der Ausgang Q sofort rueckgesetzt.
*
* Rueckgabe : Q	 		BOOL	Pulsausgang
*			  PT		UDINT	abgelaufene Pulsdauer in [10 ms]
*
* History   :
*  V1.00	  14.09.1998,fw			erstellt
*  V1.10      17.05.2002,fw     	Funktion SYS_info durch Funtionsblock SysInfo ersetzt,
*                               	damit die Library auch für i386 kompiliert werden kann.
*  V1.70	  17.06.2002,WeitzerT	inc. plctypes entf.; bei jewlib1.h <> statt ""
*
***********************************************************************************/
#include <jew_lib1.h>
#include <brsystem.h>

void TP_R(TP_R_typ *fd)
{
	SysInfo_typ	SysInf;
	unsigned long time_over;

	SysInf.enable = 1;
	SysInfo(&SysInf);

	if (fd->IN != fd->IN_old)
	{
		fd->IN_old = fd->IN;
		if (fd->IN == 1)
			fd->Q = 1;
	}

	if (fd->Q == 1)
	{
		if (SysInf.tick_count >= fd->tick_old)
			time_over = SysInf.tick_count - fd->tick_old;
		else
			time_over = 0 - fd->tick_old + SysInf.tick_count;

		fd->ET = fd->ET + time_over;

		if (fd->ET >= fd->PT)
		{
			fd->Q = 0;
			fd->ET = 0;
		}

		if (SysInf.init_count != fd->init_old)
		{
			fd->Q = 1;
			fd->ET = 0;
			fd->init_old = SysInf.init_count;
		}
	}

	if (fd->RS == 1)
	{
		fd->Q = 0;
		fd->ET = 0;
	}

	fd->tick_old = SysInf.tick_count;

}
```

#### uc_bitclr.c
```c
/***********************************************************************************
* Name      : uc_BitClr.c
* Titel     : Setzen einer Bit-Stelle eines unsigned char auf FALSE
* Version   : V1.0
* Datum     : 15.10.2001
*
* Uebergabe : In				USINT			Wert mit zu setzender Bit Stelle
*			: BitNr				USINT			Bit Stelle die gesetzt werden soll
*
* Rueckgabe : function			USINT			Wert mit gesetzter Bit Stelle
*
* History   :
*  V1.00	  15.10.2001,Fa			erstellt
*  V1.70	  17.06.2002,WeitzerT	bei jewlib1.h <> statt ""
*
***********************************************************************************/
#include <jew_lib1.h>

unsigned char uc_BitClr(unsigned char In, unsigned char BitNr)
{
	return  (In & (~(1 << BitNr)));
}
```

#### uc_bitset.c
```c
/***********************************************************************************
* Name      : uc_BitSet.c
* Titel     : Setzen einer Bit-Stelle eines unsigned char auf TRUE
* Version   : V1.0
* Datum     : 11.10.2001
*
* Uebergabe : In				USINT			Wert mit zu setzender Bit Stelle
*			: BitNr				USINT			Bit Stelle die gesetzt werden soll
*
* Rueckgabe : function			USINT			Wert mit gesetzter Bit Stelle
*
* History   :
*  V1.00	  11.10.2001,Fa			erstellt
*  V1.70	  17.06.2002,WeitzerT	bei jewlib1.h <> statt ""
*
***********************************************************************************/
#include <jew_lib1.h>

unsigned char uc_BitSet(unsigned char In, unsigned char BitNr)
{
	return  ( In | (1 << BitNr));
}
```

#### uc_bittest.c
```c
/***********************************************************************************
* Name      : uc_BitTest.c
* Titel     : Prüfen einer Bit-Stelle eines unsigned char auf TRUE
* Version   : V1.0
* Datum     : 05.09.2001
*
* Uebergabe : In				USINT			Wert mit zu püfender Bit Stelle
*			: BitNr				USINT			Bit Stelle die geprüft werden soll
*
* Rueckgabe : function			BOOL			FALSE = Bitstelle ist FALSE
*												TRUE  = Bitstelle ist TRUE
*
* History   :
*  V1.00	  05.09.2001,Fa			erstellt
*  V1.70	  17.06.2002,WeitzerT	bei jewlib1.h <> statt ""
*
***********************************************************************************/
#include <jew_lib1.h>

plcbit uc_BitTest(unsigned char In, unsigned char BitNr)
{
	return  ((In >> BitNr) & 1) != 0;
}
```

#### us_bitclr.c
```c
/***********************************************************************************
* Name      : us_BitClr.c
* Titel     : Setzen einer Bit-Stelle eines unsigned short auf FALSE
* Version   : V1.0
* Datum     : 15.10.2001
*
* Uebergabe : In				UINT			Wert mit zu setzender Bit Stelle
*			: BitNr				USINT			Bit Stelle die gesetzt werden soll
*
* Rueckgabe : function			UINT			Wert mit gesetzter Bit Stelle
*
* History   :
*  V1.00	  15.10.2001,Fa			erstellt
*  V1.70	  17.06.2002,WeitzerT	bei jewlib1.h <> statt ""
*
***********************************************************************************/
#include <jew_lib1.h>

unsigned short us_BitClr(unsigned short In, unsigned char BitNr)
{
	return  (In & (~(1 << BitNr)));
}
```

#### us_bittest.c
```c
/***********************************************************************************
* Name      : us_BitTest.c
* Titel     : Prüfen einer Bit-Stelle eines unsigned short auf TRUE
* Version   : V1.0
* Datum     : 15.09.2001
*
* Uebergabe : In				UINT			Wert mit zu püfender Bit Stelle
*			: BitNr				USINT			Bit Stelle die geprüft werden soll
*
* Rueckgabe : function			BOOL			FALSE = Bitstelle ist FALSE
*												TRUE  = Bitstelle ist TRUE
*
* History   :
*  V1.00	  15.09.2001,Fa			erstellt
*  V1.70	  17.06.2002,WeitzerT	bei jewlib1.h <> statt ""
*
***********************************************************************************/
#include <jew_lib1.h>

plcbit us_BitTest(unsigned short In, unsigned char BitNr)
{
	return  ((In >> BitNr) & 1) != 0;
}
```

#### wdtobit.c
```c
/***********************************************************************************
* Name      : WDtoBIT.c
* Titel     : Ein Word(2Byte) auf 16 Bits dekomprimieren
* Version   : V1.00
* Datum     : 09.11.1998
*
* Uebergabe : Word 		UINT	Kompriemiertes Ausgangsabbild
*
* Rueckgabe : Bit00		BOOL	Bit 00 des Eingangswortes
*			  Bit01		BOOL	Bit 01 des Eingangswortes
*			  Bit02		BOOL	Bit 02 des Eingangswortes
*			  Bit03		BOOL	Bit 03 des Eingangswortes
*			  Bit04		BOOL	Bit 04 des Eingangswortes
*			  Bit05		BOOL	Bit 05 des Eingangswortes
*			  Bit06		BOOL	Bit 06 des Eingangswortes
*			  Bit07		BOOL	Bit 07 des Eingangswortes
*			  Bit08		BOOL	Bit 08 des Eingangswortes
*			  Bit09		BOOL	Bit 09 des Eingangswortes
*			  Bit10		BOOL	Bit 10 des Eingangswortes
*			  Bit11		BOOL	Bit 11 des Eingangswortes
*			  Bit12		BOOL	Bit 12 des Eingangswortes
*			  Bit13		BOOL	Bit 13 des Eingangswortes
*			  Bit14		BOOL	Bit 14 des Eingangswortes
*			  Bit15		BOOL	Bit 15 des Eingangswortes
*
* History   :
*  V1.00	  09.11.1998,fw		erstellt
*  V1.70	  17.06.2002,WeitzerT	inc. plctypes entf.; bei jewlib1.h <> statt ""
*
***********************************************************************************/
#include <jew_lib1.h>

void WDtoBIT(WDtoBIT_typ *fd)
{
	fd->Bit00 = (fd->Word) & 1;
	fd->Bit01 = (fd->Word>>1) & 1;
	fd->Bit02 = (fd->Word>>2) & 1;
	fd->Bit03 = (fd->Word>>3) & 1;
	fd->Bit04 = (fd->Word>>4) & 1;
	fd->Bit05 = (fd->Word>>5) & 1;
	fd->Bit06 = (fd->Word>>6) & 1;
	fd->Bit07 = (fd->Word>>7) & 1;
	fd->Bit08 = (fd->Word>>8) & 1;
	fd->Bit09 = (fd->Word>>9) & 1;
	fd->Bit10 = (fd->Word>>10) & 1;
	fd->Bit11 = (fd->Word>>11) & 1;
	fd->Bit12 = (fd->Word>>12) & 1;
	fd->Bit13 = (fd->Word>>13) & 1;
	fd->Bit14 = (fd->Word>>14) & 1;
	fd->Bit15 = (fd->Word>>15) & 1;
}
```

#### xsignscal_R.c
```c
/********************************************************************
 * COPYRIGHT -- INNIO Company
 ********************************************************************
 * Library: JEW_LIB1
 * File: xsignscal_R.c
 * Author: 320003156
 * Created: August 24, 2011
 *******************************************************************/

#include <jew_lib1.h>

void xSignScal_R(xSignScal_R_typ* inst)
{
	unsigned long	usxPointNr;
	signed long		slErg;
	short*			PointAdress;

	inst->error = 0;			/* Error Bit zurücksetzen	*/
	inst->exceed= 0;
	usxPointNr = 0;

	if (inst->enable != 0)
	{
		if (inst->num > 1)
		{
			PointAdress = (short*)inst->param;
		/*	usxPointNr = inst->num;
			inst-> Out = PointAdress[usxPointNr];	*/

			/* prüfen ob In kleiner als des kleinste x-Element ist */
			if (inst->In < PointAdress[0])
			{
				inst->exceed = 1;			/* Eingabebereich unterschritten	*/
				usxPointNr 	 = 1;			/* Berechnung mit ersten Wertepaaren*/
			}
			/* prüfen ob In kleiner als des kleinste Element ist */
			else if (inst->In >= PointAdress[(inst->num <<1)-2])
			{
				usxPointNr = inst->num-1;		 /* Berechnung mit letzten Wertepaaren	*/
				if (inst->In > PointAdress[(inst->num <<1)-2])
				{
					inst->exceed = 1; 		/* Eingabebereich überschritten	*/
				}
			}
			/* suchen der Wertepaare im passenden Abschnitt	*/
			else
			{
				while (inst->In >= PointAdress[usxPointNr<<1]) usxPointNr++;
			}

			/* Berechnung mittels Geradengleichung und der ermittelten Wertepaare	*/
			usxPointNr = usxPointNr*2 - 2;		/* usxPointNr auf erstes Element der Wertepaare stellen	*/
			if (PointAdress[usxPointNr] != PointAdress[usxPointNr+2])
			{
				slErg = (inst->In - PointAdress[usxPointNr])*(PointAdress[usxPointNr+3]-PointAdress[usxPointNr+1])/(PointAdress[usxPointNr+2]-PointAdress[usxPointNr])+ PointAdress[usxPointNr+1];

				if (slErg > 32767)	inst->Out = 32767;				/* Ergebnis über Wertebereich von short */
				else if (slErg < -32768)	inst->Out = -32768;		/* Ergebnis unter Wertebereich von short*/
				else inst->Out = slErg;						/* Ergebnis ausgeben					*/
			}
			else
			{
				inst->error = 1;	/* zwei x-Werte sind gleich	*/
				inst->Out 	= 0;
			}
		}
		else
		{
			inst->error = 1;	/* mindestens zwei Wertepaare sind notwendig	*/
			inst->Out 	= 0;
		}
	}
}
```

#### xsignscal.c
```c
/***********************************************************************************
* Name      : xSignScal.c
* Titel     : Lineare Interpolation aus num Stützstellen
* Version   : V1.0
* Datum     : 21.08.2001
*
* Uebergabe : enable			BOOL			Bearbeitung des Funktionsblockes aus/ein
*			: num				UINT			Anzahl der Stützstellen
*			: param				ULONG			Adresse der Stützstellenpaare
*			: In				INT				Aktueller Analogwert
*
* Rueckgabe : error	 			BOOL			Fehlparametrierung: 0= kein Fehler, 1= Fehler
*			: Out				INT	    		Funktionsabhängiger Ausgabewert
*
* History   :
*  V1.00	  21.08.2001,Fa			erstellt
*  V1.70	  17.06.2002,WeitzerT	inc. plctypes entf.; bei jewlib1.h <> statt ""
*
***********************************************************************************/
#include <jew_lib1.h>

void xSignScal(xSignScal_typ* inst)
{
	unsigned long	usxPointNr;
	signed long		slErg;
	short*			PointAdress;

	inst->error = 0;			/* Error Bit zurücksetzen	*/
	inst->exceed= 0;
	usxPointNr = 0;

	if (inst->enable != 0)
	{
		if (inst->num > 1)
		{
			PointAdress = (short*)inst->param;
		/*	usxPointNr = inst->num;
			inst-> Out = PointAdress[usxPointNr];	*/

			/* prüfen ob In kleiner als des kleinste x-Element ist */
			if (inst->In < PointAdress[0])
			{
				inst->exceed = 1;			/* Eingabebereich unterschritten	*/
				usxPointNr 	 = 1;			/* Berechnung mit ersten Wertepaaren*/
			}
			/* prüfen ob In kleiner als des kleinste Element ist */
			else if (inst->In >= PointAdress[(inst->num <<1)-2])
			{
				usxPointNr = inst->num-1;		 /* Berechnung mit letzten Wertepaaren	*/
				if (inst->In > PointAdress[(inst->num <<1)-2])
				{
					inst->exceed = 1; 		/* Eingabebereich überschritten	*/
				}
			}
			/* suchen der Wertepaare im passenden Abschnitt	*/
			else
			{
				while (inst->In >= PointAdress[usxPointNr<<1]) usxPointNr++;
			}

			/* Berechnung mittels Geradengleichung und der ermittelten Wertepaare	*/
			usxPointNr = usxPointNr*2 - 2;		/* usxPointNr auf erstes Element der Wertepaare stellen	*/
			if (PointAdress[usxPointNr] != PointAdress[usxPointNr+2])
			{
				slErg = ((long)inst->In - PointAdress[usxPointNr])*(PointAdress[usxPointNr+3]-PointAdress[usxPointNr+1])/(PointAdress[usxPointNr+2]-PointAdress[usxPointNr])+ PointAdress[usxPointNr+1];

				if (slErg > 32767)	inst->Out = 32767;				/* Ergebnis über Wertebereich von short */
				else if (slErg < -32768)	inst->Out = -32768;		/* Ergebnis unter Wertebereich von short*/
				else inst->Out = (short)slErg;						/* Ergebnis ausgeben					*/
			}
			else
			{
				inst->error = 1;	/* zwei x-Werte sind gleich	*/
				inst->Out 	= 0;
			}
		}
		else
		{
			inst->error = 1;	/* mindestens zwei Wertepaare sind notwendig	*/
			inst->Out 	= 0;
		}
	}
}
```

#### gr_minR.c
```c
/********************************************************************
 * COPYRIGHT -- INNIO Company
 ********************************************************************
 * Library: JEW_LIB1
 * File: gr_minR.c
 * Author: 320003156
 * Created: August 17, 2011
 *******************************************************************/

#include <jew_lib1.h>

void GR_MINR(GR_MINR_typ *fd)
{
	if (fd->In <= fd->Gw)
		fd->Q = 1;
	else if (fd->In > (fd->Gw + fd->Hy))
		fd->Q = 0;
}
```

#### filter_R.c
```c
/********************************************************************
 * COPYRIGHT -- INNIO Company
 ********************************************************************
 * Library: JEW_LIB1
 * File: filter_R.c
 * Author: 320003156
 * Created: August 17, 2011
 *
 * History   :
 *  V1.91	  02.02.2022,Schmid		added Reset input
 *
*******************************************************************/

#include <jew_lib1.h>

void FILTER_R(FILTER_R_typ *fd)
{
	if (fd->Filter == 0.0)
		fd->Filter = 1.0;				/* Division durch 0 verhindern */

	if (fd->Reset)
		fd->temp_mw = fd->In * fd->Filter;
	else
		fd->temp_mw = fd->temp_mw + fd->In - fd->Out;

	fd->Out = fd->temp_mw/fd->Filter;
}
```

#### ul_bitset.c
```c
/***********************************************************************************
* Name      : ul_BitSet.c
* Titel     : Setzen einer Bit-Stelle eines unsigned long auf TRUE
* Version   : V1.0
* Datum     : 17.10.2022
*
* Uebergabe : In				UDINT			Wert mit zu setzender Bit Stelle
*			: BitNr				USINT			Bit Stelle die gesetzt werden soll
*
* Rueckgabe : function			UDINT			Wert mit gesetzter Bit Stelle
*
* History   :
*  V1.00	  17.10.2022 Racero, Guillermo     Created based on us_BitSet.c
*
***********************************************************************************/
#include <jew_lib1.h>

unsigned long ul_BitSet(unsigned long In, unsigned char BitNr)
{
	return  ( In | (1 << BitNr));
}
```

#### ul_bitclr.c
```c
/***********************************************************************************
* Name      : ul_BitClr.c
* Titel     : Setzen einer Bit-Stelle eines unsigned long auf FALSE
* Version   : V1.0
* Datum     : 17.10.2022
*
* Uebergabe : In				UDINT			Wert mit zu setzender Bit Stelle
*			: BitNr				USINT			Bit Stelle die gesetzt werden soll
*
* Rueckgabe : function			UDINT			Wert mit gesetzter Bit Stelle
*
* History   :
*  V1.00	  17.10.2022 Racero, Guillermo     Created based on us_BitClr.c
*
***********************************************************************************/
#include <jew_lib1.h>

unsigned long ul_BitClr(unsigned long In, unsigned char BitNr)
{
	return  (In & (~(1 << BitNr)));
}
```

#### ul_bittest.c
```c
/***********************************************************************************
* Name      : ul_BitTest.c
* Titel     : Prüfen einer Bit-Stelle eines unsigned long auf TRUE
* Version   : V1.0
* Datum     : 09.12.2022
*
* Uebergabe : In				UDINT			Wert mit zu püfender Bit Stelle
*			: BitNr				USINT			Bit Stelle die geprüft werden soll
*
* Rueckgabe : function			BOOL			FALSE = Bitstelle ist FALSE
*												TRUE  = Bitstelle ist TRUE
*
* History   :
* V1.0	09.12.2022	Andre,	Created based on us_BitTest.c
*
***********************************************************************************/
#include <jew_lib1.h>

plcbit ul_BitTest(unsigned long In, unsigned char BitNr)
{
	return  ((In >> BitNr) & 1) != 0;
}
```

### Library Logical/Libraries/JWASLIB2 (ANSIC, version 2.00.0)

#### JWASLIB2.fun
```iecst
FUNCTION xornt_16b : INT
	VAR_INPUT
		I1 : UDINT;
		I2N : UDINT;
		Q : UDINT;
	END_VAR
END_FUNCTION

FUNCTION sum_16b : INT
	VAR_INPUT
		IN : UDINT;
	END_VAR
END_FUNCTION

FUNCTION xor_16b : INT
	VAR_INPUT
		I1 : UDINT;
		I2 : UDINT;
		Q : UDINT;
	END_VAR
END_FUNCTION

FUNCTION_BLOCK AmmSequence
	VAR_INPUT
		Enable : BOOL;
		ClockPulse : BOOL;
		NrOfBits : USINT;
		BitArray : UDINT;
	END_VAR
	VAR_OUTPUT
		Alarm1 : BOOL;
		Alarm2 : BOOL;
		ErrorNr : USINT;
		Status : UINT;
	END_VAR
	VAR
		InputArray : ARRAY[0..255] OF BOOL;
		OutputArray : ARRAY[0..255] OF BOOL;
		ChkValue : USINT;
		ChkEdge : BOOL;
	END_VAR
END_FUNCTION_BLOCK

FUNCTION polyg_5l : REAL
	VAR_INPUT
		x : REAL;
		coord : UDINT;
	END_VAR
END_FUNCTION

FUNCTION polyg_3hl : REAL
	VAR_INPUT
		x : REAL;
		coord : UDINT;
	END_VAR
END_FUNCTION

FUNCTION ornt_16b : INT
	VAR_INPUT
		I1 : UDINT;
		I2N : UDINT;
		Q : UDINT;
	END_VAR
END_FUNCTION

FUNCTION or_16b : INT
	VAR_INPUT
		I1 : UDINT;
		I2 : UDINT;
		Q : UDINT;
	END_VAR
END_FUNCTION

FUNCTION not_16b : INT
	VAR_INPUT
		IN : UDINT;
		Q : UDINT;
	END_VAR
END_FUNCTION

FUNCTION min_i_16b : INT
	VAR_INPUT
		IN : UDINT;
	END_VAR
END_FUNCTION

FUNCTION min_b_16b : INT
	VAR_INPUT
		IN : UDINT;
		Q : UDINT;
	END_VAR
END_FUNCTION

FUNCTION min_16di : INT
	VAR_INPUT
		EN : UDINT;
		IN : UDINT;
		Q : UDINT;
	END_VAR
END_FUNCTION

FUNCTION max_i_16b : INT
	VAR_INPUT
		IN : UDINT;
	END_VAR
END_FUNCTION

FUNCTION max_b_16b : INT
	VAR_INPUT
		IN : UDINT;
		Q : UDINT;
	END_VAR
END_FUNCTION

FUNCTION max_16di : INT
	VAR_INPUT
		EN : UDINT;
		IN : UDINT;
		Q : UDINT;
	END_VAR
END_FUNCTION

FUNCTION i32_t_i16 : INT
	VAR_INPUT
		IN : DINT;
	END_VAR
END_FUNCTION

FUNCTION compr_16b : INT
	VAR_INPUT
		IN : UDINT;
		Q : UDINT;
	END_VAR
END_FUNCTION

FUNCTION andnt_16b : INT
	VAR_INPUT
		I1 : UDINT;
		I2N : UDINT;
		Q : UDINT;
	END_VAR
END_FUNCTION

FUNCTION and_16b : INT
	VAR_INPUT
		I1 : UDINT;
		I2 : UDINT;
		Q : UDINT;
	END_VAR
END_FUNCTION

FUNCTION polyg_2hl : REAL
	VAR_INPUT
		x : REAL;
		coord : UDINT;
	END_VAR
END_FUNCTION
```

#### JWASLIB2.var
```iecst
VAR CONSTANT
	AMM_SEQ_ERROR_NO_ARRAY_ADDRESS	: UINT	:= 1;
	AMM_SEQ_ERROR_NO_ARRAY_LENGTH	: UINT	:= 2;
END_VAR
```

#### JWASLIB2.typ
```iecst
(********************************************************************
 * COPYRIGHT -- INNIO Company
 ********************************************************************
 * Library: JWASLIB2
 * File: JWASLIB2.typ
 * Author: 105051626
 * Created: February 04, 2014
 ********************************************************************
 * Data types of library JWASLIB2
 ********************************************************************)

TYPE
	coordinate_5 : 	STRUCT
		x1 : REAL;
		x2 : REAL;
		x3 : REAL;
		x4 : REAL;
		x5 : REAL;
		y1 : REAL;
		y2 : REAL;
		y3 : REAL;
		y4 : REAL;
		y5 : REAL;
	END_STRUCT;
	IntegralElement : 	STRUCT
		In : REAL;
		In_internal : REAL;
		In_ref : REAL;
		mode : INT;
		Ki_plus : REAL;
		Ki_minus : REAL;
		dOut_plus : REAL;
		dOut_minus : REAL;
		dOut_max_p : REAL;
		dOut_max_m : REAL;
		Out_min : REAL;
		Out_max : REAL;
		Out_internal : REAL;
		Out : REAL;
	END_STRUCT;
	IntegralController : 	STRUCT
		enable : BOOL;
		x : REAL;
		w : REAL;
		w_ref : REAL;
		mode : INT;
		deadband : REAL;
		Ki_plus : REAL;
		Ki_minus : REAL;
		dy_plus : REAL;
		dy_minus : REAL;
		dy_max_p : REAL;
		dy_max_m : REAL;
		y_block : REAL;
		y_min : REAL;
		y_max : REAL;
		y_invers : BOOL;
		y_internal : REAL;
		y : REAL;
	END_STRUCT;
END_TYPE
```

#### amm_seq.c
```c
/***********************************************************************************
* Name      : JWASLIB2
* Title     : Special functions for module controll
* Version   : V1.40
* Date      : 18.02.2004
*
* History   :
*  V1.40	  18.02.2004,TEE/TW add function block AlarmSequence
*  V1.41	  16.12.2004,TEE/TW AmmSequence: alarm reset handling improved
*
*
***********************************************************************************/
/*******************************************************************************
* AGGR: AmmSequence.c - message sequencer for alarm management
*
* This code is confidential and proprietary to the INNIO Company.
* It may not be used in any form, or reproduced in any manner, without the express
* written permission of the INNIO Company.
* Copyright, INNIO Company, 2004
*
* Input : 	Enable		BOOL		enable function block
*			ClockPulse	BOOL		external clock pulse to sequence the different amm messages (AM)
*			NrOfBits	USINT		number of bits that should be checked
*			BitArray	UDINT		address of the alram bit array
*
* Output:   Alarm1		BOOL		if any AM in the array is active then the output is 1
*           Alarm2		BOOL		signals the output of a new AM with the same pulse as the clock pulse
*			ErrorNr		USINT		signals the bit number of a new AM
*			Status		UINT		gives back a number if fub works correct or not
*
* Var	:	InputArray	BOOL[256]	image of input array
*			OutputArray BOOL[256]	image of output array
*			ChkValue	USINT		check counter for sequencing
*			ChkEdge		BOOL		check the rising edge of the pulse signal
*
* History:
* -------
* V0.1	18-02-04	Weitzer, generated
*
* V0.2	16-12-04	Weitzer, alarm reset handling improved
*
* V0.3	02-11-05	Weitzer, reset of Alarm1 and Alarm2 bits if inputs and enable is false
*
* Outstandings:
* ------------
*
*******************************************************************************/
#include <JWASLIB2.h>

void AmmSequence(AmmSequence_typ* inst)
{

	/* declaration of additional tags */

	unsigned short	n;				/* counter for loops */
	unsigned short	InputSum;		/* check if any alarm is set */
	plcbit*			ArrayAdr;		/* data tag for adress pointer */
	plcbit			ResetAll;		/* flag for erasing all entries */

	/* prepare data copy from bit array address */

	ArrayAdr = (plcbit*)inst->BitArray;

	/* check if FUB is enabled to run */

	if(inst->Enable != 1)
	{

		/* check if all alarms were put out or a alarm was gone */
		ResetAll = 0;
		InputSum = 0;
		for(n = 0; n < inst->NrOfBits; ++n)		/* loop over the complete bit array */
		{
			/* check if data adress is valid and for diffences between input and output array */
			if (ArrayAdr != 0)
			{
				if (inst->OutputArray[n] != ArrayAdr[n])	ResetAll = 1;		/* set reset flag */
				InputSum = InputSum + ArrayAdr[n];								/* check if any error is set */
			}
		}

		/* if reset flag was set -> reset data = acknowledgement */
		if (ResetAll == 1 || InputSum == 0)
		{
			inst->Alarm1   = 0;		/* reset alarm output 1 */
			inst->Alarm2   = 0;		/* reset alarm output 2 */
			inst->ErrorNr  = 0;		/* reset error number output */
			inst->ChkValue = 0;		/* reset check value */
			inst->ChkEdge  = 0;		/* reset check edge */

			for(n = 0; n < inst->NrOfBits; ++n)		/* loop over the complete bit array */
			{
				inst->InputArray[n]  = 0;		/* reset image of input array  */
				inst->OutputArray[n] = 0;		/* reset image of output array */
			}
		}
		inst->Status   = 0;		/* reset status output */

	}

	/* if FUB is enabled -> monitoring and output is active */
	else
	{

		/* check if address of bit array exists */
		if(ArrayAdr != 0)
		{

			/* search in the array for new alarm messages */

			for(n = 0; n < inst->NrOfBits; ++n)		/* loop over the number of bits */
			{
				/* check bit array address at position n */
				if(ArrayAdr[n] == 1)
				{
			 		/* check if it is the first entry */
					if(inst->Alarm1 == 0)
					{
						inst->ErrorNr  = n;			/* set output error number */
						inst->ChkValue = 0;			/* reset check value to start with number output */
					}
					inst->Alarm1        = 1;		/* set general alarm output 1 */
					inst->InputArray[n] = 1;		/* set alarm entry at the input image */
				}
			}

			/* create sequenced alarm output */

			/* if any entry has been made */
			if(inst->Alarm1 == 1)
			{
				/* wait for positiv edge of the pulse input */
				if(inst->ClockPulse == 1)
				{
					/* check if it was the first call after the edge */
					if(inst->ChkEdge == 0)
					{
						inst->ChkEdge = 1;		/* set check bit for toggeling the check value */

						/* toggeling between number and pulse output */

						/* number output */
						if(inst->ChkValue == 0)
						{
							for(n = 0; n < inst->NrOfBits; ++n)		/* loop over the number of bits */
							{
								/* check for alarm message which were not copied to the output entry */
								if(inst->OutputArray[n] == 0)
								{
									/* set output if there is a new message in the input image */
									if(inst->InputArray[n] == 1)
									{
										inst->Alarm2         = 0;					/* set alarm output pulse */
										inst->ErrorNr        = n;					/* set output error number */
										inst->OutputArray[n] = 1;					/* set entry in the output image */
										n                    = inst->NrOfBits;		/* exit loop */
										inst->ChkValue       = 1;					/* set value to detect the change */
									}
								}

								/* check bit array at position n if inputs have gone */
								else if (ArrayAdr[n] == 0) inst->InputArray[n]  = 0;		/* reset entry in the input image */

								/* check if old messages exits */
								inst->ChkValue = inst->ChkValue + inst->OutputArray[n];
							}

							/* check if no new message or no old message exits */
							if(inst->ChkValue == 0)
							{
								inst->Alarm1 = 0;		/* reset alarm output 1 if no alarm in the input image */
								inst->Alarm2 = 0;		/* reset alarm output pulse if no alarm to output */
							}
							else inst->ChkValue = 1;		/* else output next message */

						}

						/* pulse output Alarm2 */
						else
						{
							inst->Alarm2   = 1;		/* set alarm output pulse */
							inst->ChkValue = 0;		/* reset check value for switching to pulse output */
						}
					}
				}
				else inst->ChkEdge = 0;		/* reset edge detection */
			}

		}

		/* error handling */

		/* set status output to 1 if no pointer connected */
		else inst->Status  = 1;

		/* set status output to 2 if number of bits is 0 */
		if(inst->NrOfBits == 0) inst->Status = 2;
	}
}
```

#### functions1.c
```c
/***********************************************************************************
* Name      : jwaslib2
* Titel     : Sonderfunktionen erstellt für Modulsteuerung
* Version   : V1.40
* Datum     : 18.02.2004
*
* History   :
*  V1.00	  23.12.1998,fw		erstellt
*  V1.20	  14.04.1999,fw		neue Funktionen, ueberarbeiten der alten Funktionen
*  V1.31	  24.09.2003,TEE/TW Einbindung in Librarymanager
*  V1.40	  18.02.2004,TEE/TW Neue Funktionsblock AlarmSequence unter amm_seq.c hinzugefügt
*  V1.50	  08.08.2017,FW Für GCC 4.1.2 adaptiert
*  V2.00    26.06.2018,FW, datatype changed from signed short to float in polygon FUBs
*
* Hinweis	: Bei der Strukturdefinition ist folgendes zu beachten:
* 				Alle nicht-boolschen Elemente eines FUB muessen vor den boolschen
*				Elementen in der Reihenfolge Input, Output, Statisch definiert werden.
*
***********************************************************************************/

#include <bur/plc.h>
#include <bur/plctypes.h>
#include <JWASLIB2.h>

/***********************************************************************************
* AND for data type ARRAY OF 16 BOOL
* Copyright 1998 - 1999 Jenbacher Werke AG
*
* History:
* -------
* V0.1	01-04-99	Thaler, generated from FB219
* V1.50 08-08-2017  FW, adapted for GCC 4.1.2
*
* Outstandings:
* ------------
*
***********************************************************************************/
signed short and_16b(UDINT I1, UDINT I2, UDINT Q)
{
	signed short	x;
	BOOL *i1, *i2, *q;

	i1 = (BOOL*)I1;
	i2 = (BOOL*)I2;
	q = (BOOL*)Q;

	for (x=1; x<=16; x++)
		q[x] = i1[x] & i2[x];
	return 0;
}

/*******************************************************************************
* AND NOT for data type ARRAY OF 16 BOOL
* Copyright 1998 - 1999 Jenbacher Werke AG
*
* History:
* -------
* V0.1	01-04-99	Thaler, generated from FB220
*		13-04-99	Thaler, name changed
* V1.50 08-08-2017  FW, adapted for GCC 4.1.2
*
* Outstandings:
* ------------
*
*******************************************************************************/
signed short andnt_16b(UDINT I1, UDINT I2N, UDINT Q)
{
	signed short	x;
	BOOL *i1, *i2n, *q;

	i1 = (BOOL*)I1;
	i2n = (BOOL*)I2N;
	q = (BOOL*)Q;

	for (x=1; x<=16; x++)
		q[x] = i1[x] & !i2n[x];
	return 0;
}

/*******************************************************************************
* Compress an ARRAY OF 16 BOOL
* Copyright 1998 - 1999 Jenbacher Werke AG
*
* History:
* -------
* V0.1	01-04-99	Thaler, generated from FB192
* V1.50 08-08-2017  FW, adapted for GCC 4.1.2
*
* Outstandings:
* ------------
*
*******************************************************************************/
signed short compr_16b(UDINT IN, UDINT Q)
{
	signed short	a, x;
	BOOL	*in, *q;

	in = (BOOL*)IN;
	q = (BOOL*)Q;

	for (x=1; x<=16; x++)
		q[x] = 0;

	a = 1;

	for (x=1; x<=16; x++)
	{
		if (in[x])
		{
			q[a] = 1;
			a++;
		}
	}
	return 0;
}

/*******************************************************************************
* Type conversion with min- / max-limitation
* Copyright 1998 - 1999 Jenbacher AG
*
* History:
* -------
* V0.1	31-03-99	Thaler, generated from FB200
*		13-04-99	Thaler, name changed
* V0.2
*
* Outstandings:
* ------------
*
*******************************************************************************/
signed short i32_t_i16(signed long IN)
{
	signed long	mn = -32768;
	signed long	mx = 32767;

	if (IN < mn)
		IN = mn;
	else if (IN > mx)
		IN = mx;

	return (short)(IN);
}

/*******************************************************************************
* Max input channel of an ARRAY OF 16 DINT, result as BOOL
* Copyright 1998 - 1999 Jenbacher AG
*
* History:
* -------
* V0.1	01-04-99	Thaler, generated from FB207
* V1.50 08-08-2017  FW, adapted for GCC 4.1.2
*
* Outstandings:
* ------------
*
*******************************************************************************/
signed short max_16di(UDINT EN, UDINT IN, UDINT Q)
{
	signed short	x;
	signed short	b = 0;
	signed long		d = 0x80000000;
	BOOL	*en, *q;
	DINT	*in;

	en = (BOOL*)EN;
	in = (DINT*)IN;
	q = (BOOL*)Q;

	for (x=1; x<=16; x++)
		q[x] = 0;

	for (x=1; x<=16; x++)
	{
		if (en[x])
		{
			if (in[x] >= d)
			{
				d = in[x];
				b = x;
			}
		}
	}

	q[b] = 1;
	return 0;
}

/*******************************************************************************
* Max input channel of an ARRAY OF 16 BOOL, result as BOOL
* Copyright 1998 - 1999 Jenbacher Werke AG
*
* History:
* -------
* V0.1	01-04-99	Thaler, generated
* V1.50 08-08-2017  FW, adapted for GCC 4.1.2
*
* Outstandings:
* ------------
*
*******************************************************************************/
signed short max_b_16b(UDINT IN, UDINT Q)
{
	signed short	x;
	BOOL	*in, *q;

	in = (BOOL*)IN;
	q = (BOOL*)Q;

	for (x=1; x<=16; x++)
		q[x] = 0;

	x = 16;
	while ((in[x]==0) && (x!=0))
		x--;

	if (x)
		q[x] = 1;
	return 0;
}

/*******************************************************************************
* Max input channel of an ARRAY OF 16 BOOL, result as INT
* Copyright 1998 - 1999 Jenbacher Werke AG
*
* History:
* -------
* V0.1	16-11-98	Thaler, generated from FB222
*		02-04-99	Thaler, name of VAR_INPUT modified
* V1.50 08-08-2017  FW, adapted for GCC 4.1.2
*
* Outstandings:
* ------------
*
*******************************************************************************/
signed short max_i_16b(UDINT IN)
{
	signed short	x;
	signed short	MAX_I_16b = 0;
	BOOL	*in;

	in = (BOOL*)IN;

	for (x=1; x<=16; x++)
	{
		if (in[x])
		{
			MAX_I_16b = x;
		}
	}
	return MAX_I_16b;
}
/*******************************************************************************
* Min input channel of an ARRAY OF 16 DINT, result as BOOL
* Copyright 1998 - 1999 Jenbacher AG
*
* History:
* -------
* V0.1	01-04-99	Thaler, generated from FB207
* V1.50 08-08-2017  FW, adapted for GCC 4.1.2
*
* Outstandings:
* ------------
*
*******************************************************************************/
signed short min_16di(UDINT EN, UDINT IN, UDINT Q)
{
	signed short	x;
	signed short	b = 0;
	signed long		d = 0x7FFFFFFF;
	BOOL	*en, *q;
	DINT	*in;

	en = (BOOL*)EN;
	in = (DINT*)IN;
	q = (BOOL*)Q;

	for (x=1; x<=16; x++)
		q[x] = 0;

	for (x=1; x<=16; x++)
	{
		if (en[x])
		{
			if (in[x] <= d)
			{
				d = in[x];
				b = x;
			}
		}
	}

	q[b] = 1;
	return 0;
}

/*******************************************************************************
* Min input channel of an ARRAY OF 16 BOOL, result as BOOL
* Copyright 1998 - 1999 Jenbacher Werke AG
*
* History:
* -------
* V0.1	01-04-99	Thaler, generated from FB191
* V1.50 08-08-2017  FW, adapted for GCC 4.1.2
*
* Outstandings:
* ------------
*
*******************************************************************************/
signed short min_b_16b(UDINT IN, UDINT Q)
{
	signed short	x;
	BOOL	*in, *q;

	in = (BOOL*)IN;
	q = (BOOL*)Q;

	for (x=1; x<=16; x++)
		q[x] = 0;

	for (x=1; x<=16; x++)
	{
		if (in[x])
		{
			q[x] = 1;
			break;
		}
	}
	return 0;
}

/*******************************************************************************
* Min input channel of an ARRAY OF 16 BOOL, result as INT
* Copyright 1998 - 1999 Jenbacher Werke AG
*
* History:
* -------
* V0.1	16-11-98	Thaler, generated from FB222
*		02-04-99	Thaler, name of VAR_INPUT modified
* V1.50 08-08-2017  FW, adapted for GCC 4.1.2
*
* Outstandings:
* ------------
*
*******************************************************************************/
signed short min_i_16b(UDINT IN)
{
	signed short	x;
	signed short	MIN_I_16b = 0;
	BOOL	*in;

	in = (BOOL*)IN;

	for (x=1; x<=16; x++)
	{
		if (in[x])
		{
			MIN_I_16b = x;
			break;
		}
	}
	return MIN_I_16b;
}

/*******************************************************************************
* NOT for data type ARRAY OF 16 BOOL
* Copyright 1998 - 1999 Jenbacher Werke AG
*
* History:
* -------
* V0.1	01-04-99	Thaler, generated
* V1.50 08-08-2017  FW, adapted for GCC 4.1.2
*
* Outstandings:
* ------------
*
*******************************************************************************/
signed short not_16b(UDINT IN, UDINT Q)
{
	signed short	x;
	BOOL	*in, *q;

	in = (BOOL*)IN;
	q = (BOOL*)Q;

	for (x=1; x<=16; x++)
		q[x] = !in[x];
	return 0;
}

/*******************************************************************************
* OR for data type ARRAY OF 16 BOOL
* Copyright 1998 - 1999 Jenbacher Werke AG
*
* History:
* -------
* V0.1	01-04-99	Thaler, generated
* V1.50 08-08-2017  FW, adapted for GCC 4.1.2
*
* Outstandings:
* ------------
*
*******************************************************************************/
signed short or_16b(UDINT I1, UDINT I2, UDINT Q)
{
	signed short	x;
	BOOL *i1, *i2, *q;

	i1 = (BOOL*)I1;
	i2 = (BOOL*)I2;
	q = (BOOL*)Q;

	for (x=1; x<=16; x++)
		q[x] = i1[x] | i2[x];
	return 0;
}

/*******************************************************************************
* OR NOT for data type ARRAY OF 16 BOOL
* Copyright 1998 - 1999 Jenbacher Werke AG
*
* History:
* -------
* V0.1	02-04-99	Thaler, generated
*		13-04-99	Thaler, name changed
* V1.50 08-08-2017  FW, adapted for GCC 4.1.2
*
* Outstandings:
* ------------
*
*******************************************************************************/
signed short ornt_16b(UDINT I1, UDINT I2N, UDINT Q)
{
	signed short	x;
	BOOL *i1, *i2n, *q;

	i1 = (BOOL*)I1;
	i2n = (BOOL*)I2N;
	q = (BOOL*)Q;

	for (x=1; x<=16; x++)
		q[x] = i1[x] | !i2n[x];
	return 0;
}

/*******************************************************************************
* Characteristic: polygon with 2 angles, high_limitation , low_limitation
*                 conditions: x1 < x2
*
*          y |
*            |
*         y2 +          .****
*            |        .
*            |      .
*         y1 + ****
*            |
*            +----+------+----
*                 x1     x2  x
*
* Copyright 1998 - 1999 Jenbacher AG
*
* History:
* -------
* V0.1	07-04-99	Thaler, generated from FB230
*		13-04-99	Thaler, name changed
* V1.50 08-08-2017  FW, adapted for GCC 4.1.2
* V2.00 26-06-2018  FW, datatypes of function changed from signed short to float
*
* Outstandings:
* ------------
*
*******************************************************************************/
float polyg_2hl(float x, UDINT coord)
{
	float		xL, xH, yL, yH, y;
	float		a, d;
	signed long		mn = -32768;
	signed long		mx = 32767;
	coordinate_5	*COORD;

	COORD = (coordinate_5*)coord;

	xL = COORD->x1;
	xH = COORD->x2;
	yL = COORD->y1;
	yH = COORD->y2;

	if (x <= xL)
		y = yL;
	else if (x >= xH)
		y = yH;
	else
	{
		a = (yH - yL) * (x - xL);
		if (xH != xL)
			d = yL + a / (xH - xL);
		else
			d = yL;
		/* min/max limitation */
		if (d < mn)
			d = mn;
		else if (d > mx)
			d = mx;

		y = d;
	}
	return y;
}

/*******************************************************************************
* Characteristic: polygon with 3 angles, high_limitation, low_limitation
*                 conditions: x1 < x2 < x3
*
*          y |
*            |
*         y3 +          .****
*         :  |        .
*         :  |      .
*         y1 + ****
*            |
*            +----+------+----
*                 x1 ... x3  x
*
* Copyright 1998 - 1999 Jenbacher AG
*
* History:
* -------
* V0.1	07-04-99	Thaler, generated from FB43
*		13-04-99	Thaler, name changed
* V1.50 08-08-2017  FW, adapted for GCC 4.1.2
* V2.00 26-06-2018  FW, datatypes of function changed from signed short to float
*
* Outstandings:
* ------------
*
*******************************************************************************/
float polyg_3hl(float x, UDINT coord)
{
	float			xL, xH, yL, yH, y;
	float			a, d;
	signed long		mn = -32768;
	signed long		mx = 32767;
	coordinate_5	*COORD;

	COORD = (coordinate_5*)coord;

	if (x >= COORD->x2)
	{
		xL = COORD->x2;
		xH = COORD->x3;
		yL = COORD->y2;
		yH = COORD->y3;
	}
	else
	{
		xL = COORD->x1;
		xH = COORD->x2;
		yL = COORD->y1;
		yH = COORD->y2;
	}

	if (x <= xL)
		y = yL;
	else if (x >= xH)
		y = yH;
	else
	{
		a = (yH - yL) * (x - xL);
		if (xH != xL)
			d = yL + a / (xH - xL);
		else
			d = yL;
		/* min/max limitation */
		if (d < mn)
			d = mn;
		else if (d > mx)
			d = mx;

		y = d;
	}
	return y;
}

/*******************************************************************************
* Characteristic: polygon with 5 angles, low_limitation
*                 conditions: x1 < x2 < x3 < x4 < x5
*
*          y |              .
*            |            .
*         y5 +          .
*         :  |        .
*         :  |      .
*         y1 + ****
*            |
*            +----+------+----
*                 x1 ... x5  x
*
* Copyright 1998 - 1999 Jenbacher AG
*
* History:
* -------
* V0.1	07-04-99	Thaler, generated from FB42
*		13-04-99	Thaler, name changed
* V1.50 08-08-2017  FW, adapted for GCC 4.1.2
* V2.00 26-06-2018  FW, datatypes of function changed from signed short to float
*
* Outstandings:
* ------------
*
*******************************************************************************/
float polyg_5l(float x, UDINT coord)
{
	float			xL, xH, yL, yH, y;
	float			a, d;
	signed long		mn = -32768;
	signed long		mx = 32767;
	coordinate_5	*COORD;

	COORD = (coordinate_5*)coord;

	if (x >= COORD->x4)
	{
		xL = COORD->x4;
		xH = COORD->x5;
		yL = COORD->y4;
		yH = COORD->y5;
	}
	else if (x >= COORD->x3 && x < COORD->x4)
	{
		xL = COORD->x3;
		xH = COORD->x4;
		yL = COORD->y3;
		yH = COORD->y4;
	}
	else if (x >= COORD->x2 && x < COORD->x3)
	{
		xL = COORD->x2;
		xH = COORD->x3;
		yL = COORD->y2;
		yH = COORD->y3;
	}
	else
	{
		xL = COORD->x1;
		xH = COORD->x2;
		yL = COORD->y1;
		yH = COORD->y2;
	}

	if (x <= xL)
		y = yL;
	else
	{
		a = (yH - yL) * (x - xL);
		if (xH != xL)
			d = yL + a / (xH - xL);
		else
			d = yL;
		/* min/max limitation */
		if (d < mn)
			d = mn;
		else if (d > mx)
			d = mx;

		y = d;
	}
	return y;
}

/*******************************************************************************
* Sum across an ARRAY OF 16 BOOL
* Copyright 1998 - 1999 Jenbacher Werke AG
*
* History:
* -------
* V0.1	16-11-98	Thaler, generated from FB206
*		02-04-99	Thaler, name of VAR_INPUT modified
* V1.50 08-08-2017  FW, adapted for GCC 4.1.2
*
* Outstandings:
* ------------
*
*******************************************************************************/
signed short sum_16b(UDINT IN)
{
	signed short	x;
	signed short	SUM_16b = 0;
	BOOL	*in;

	in = (BOOL*)IN;

	for (x=1; x<=16; x++)
	{
		if (in[x])
		{
			SUM_16b = SUM_16b + 1;
		}
	}
	return SUM_16b;
}

/*******************************************************************************
* XOR for data type ARRAY OF 16 BOOL
* Copyright 1998 - 1999 Jenbacher Werke AG
*
* History:
* -------
* V0.1	01-04-99	Thaler, generated
* V1.50 08-08-2017  FW, adapted for GCC 4.1.2
*
* Outstandings:
* ------------
*
*******************************************************************************/
signed short xor_16b(UDINT I1, UDINT I2, UDINT Q)
{
	signed short	x;
	BOOL *i1, *i2, *q;

	i1 = (BOOL*)I1;
	i2 = (BOOL*)I2;
	q = (BOOL*)Q;

	for (x=1; x<=16; x++)
		q[x] = i1[x] ^ i2[x];
	return 0;
}

/*******************************************************************************
* XOR NOT for data type ARRAY OF 16 BOOL
* Copyright 1998 - 1999 Jenbacher Werke AG
*
* History:
* -------
* V0.1	02-04-99	Thaler, generated
*		13-04-99	Thaler, name changed
* V1.50 08-08-2017  FW, adapted for GCC 4.1.2
*
* Outstandings:
* ------------
*
*******************************************************************************/
signed short xornt_16b(UDINT I1, UDINT I2N, UDINT Q)
{
	signed short	x;
	BOOL *i1, *i2n, *q;

	i1 = (BOOL*)I1;
	i2n = (BOOL*)I2N;
	q = (BOOL*)Q;

	for (x=1; x<=16; x++)
		q[x] = i1[x] ^ !i2n[x];
	return 0;
}
```

### Library Logical/Libraries/JWASLIB3 (ANSIC, version 0.70.0)

#### JWASLIB3.fun
```iecst
FUNCTION_BLOCK xPISchr
	VAR_INPUT
		bPIDinit	:BOOL;
		slK	:DINT;
		slTI	:DINT;
		ssW	:INT;
		ssX	:INT;
		slXWka	:DINT;
	END_VAR
	VAR_OUTPUT
		ssdY	:INT;
		slA_XWka	:DINT;
	END_VAR
END_FUNCTION_BLOCK

FUNCTION_BLOCK xPISchr_R
	VAR_INPUT
		bPIDinit	:BOOL;
		slK	:REAL;
		slTI	:REAL;
		ssW	:REAL;
		ssX	:REAL;
		slXWka	:REAL;
	END_VAR
	VAR_OUTPUT
		ssdY	:REAL;
		slA_XWka	:REAL;
	END_VAR
END_FUNCTION_BLOCK

FUNCTION_BLOCK xSigScal
	VAR_INPUT
		X	:INT;
		X1	:INT;
		Y1	:INT;
		X2	:INT;
		Y2	:INT;
	END_VAR
	VAR_OUTPUT
		Y_SCAL	:INT;
		ERROR	:BOOL;
		RUN	:BOOL;
	END_VAR
END_FUNCTION_BLOCK

FUNCTION_BLOCK xSigScal_R
	VAR_INPUT
		X	:REAL;
		X1	:REAL;
		Y1	:REAL;
		X2	:REAL;
		Y2	:REAL;
	END_VAR
	VAR_OUTPUT
		Y_SCAL	:REAL;
		ERROR	:BOOL;
		RUN	:BOOL;
	END_VAR
END_FUNCTION_BLOCK
```

#### functions.c
```c
/**************************************************************
*  functions.c - Sourcefile fuer Jenbacher-Library JWASLIB3
*  Copyright 1998 Jenbacher Werke AG
*
*  Entwicklungsgeschichte
*  ----------------------
*  V0.1   06-10-98,BrunnerK    erstellt
*  V0.2   07-08-98,BrunnerK	   FUB xSigScal geaendert
*  V0.3   11-11-98,BrunnerK    FUB xSigScal korrigiert
*  V0.4   21-01-99,FahringerA  FUB xSigScal korrigiert
*  V0.5   18-07-00,BrunnerK	   Parameter geaendert (AS V1.4 - LibManager)
*							   define´s aus h-File importiert
*  V0.6	  17-06-02,WeitzerT    include Befehle geändert
*							   (<bur/plc.h> entfernt und bei jwaslib3.h <> statt "")
*  V0.7   22-04-02,WeitzerT    Fehler bei x<x1 behoben
*  V0.7.1 24-01-14,WeitzerT	   correction of compiler warnings
*
*  Offene Punkte
*  -------------
*
***************************************************************/

#include <JWASLIB3.h>

#define vxSigMax(a,b)	((a)>(b))?(a):(b)					/* Begrenzung auf Obergrenze	*/
#define vxSigMin(a,b)	((a)<(b))?(a):(b)					/* Begrenzung auf Untergrenze 	*/
#define vxSigBet(a,b,c)	(vxSigMax((vxSigMin((c),(b))),(a)))	/* a=unterer-, c=oberer-Grenzwert	*/

/**************************************************************
*
*  Zweck:  Signalskalierung ueber Gerade (2 Punkte)
*
*  Aufruf: xSigScal(xSigScal_typ *tSigScalVar)
*
*  Übergabep.:    xSigScal_typ-Variable:
*                 X1		1. X-Koordinate
*                 Y1		1. Y-Koordinate
*                 X2		2. X-Koordinate
*                 Y2		2. Y-Koordinate
*                 X			Rohwert
*
*  Rückgabep.:    Y_SCAL	skalierter Wert
*                 RUN      	FUB in Bearbeitung
*                 ERROR     FUB-Fehler steht an
*
*  Beschreibung:  Der FUB skaliert den am Eingang anliegenden
*                 Rohwert ueber eine 2-Punkte-Gerade (x1,y1-x2,y2)
*                 Bei Bereichsueberlauf Begrenzung auf
*                 Max/Min-Wert, setzen des Error-Bits.
*
*
*
*  Datum/Autor:
*  V0.1   06-10-98,BrunnerK    erstellt
*  V0.2	  07-08-98,BrunnerK    Begrenzung auf y1 bzw. y2 eingebaut
*  V0.3   11-11-98,BrunnerK    Fehler in Berechnung behoben (fK gecastet)
*  V0.4   21-01-99,FahringerA  Float-Berechnung entfernt
*  V0.5   18-07-00,BrunnerK	   Parameter geaendert (AS V1.4 - LibManager)
*  V0.6	  17-06-02,WeitzerT    include Befehle geändert
*							   (<bur/plc.h> entfernt und bei jwaslib3.h <> statt "")
*
**************************************************************/

void xSigScal(xSigScal_typ *tSigScalVar)
{
	long	slZwischen;

	tSigScalVar->RUN = 1;
	if (tSigScalVar->X2 != tSigScalVar->X1)
	{
		tSigScalVar->ERROR  = 0;

	    /*----------------------------------------------------------*
    	* Berechnung der Skalierung                                 *
	    * Ableitung:    y = k * x + d                               *
    	*                                                           *
	    *               k = (y2-y1) / (x2-x1)                       *
    	*               d = (y1*x2 - y2*x1) / (x2-x1)               *
	    *           ==> y = (x*(y2-y1) + y1*x2 - y2*x1) / (x2-x1)   *
    	*-----------------------------------------------------------*/
    	/* Typkonvertierung auf 32Bit durchführen					*/

		slZwischen = ((tSigScalVar->X * ((long)tSigScalVar->Y2-tSigScalVar->Y1) +
					  		   ((long)tSigScalVar->Y1*tSigScalVar->X2) -
					  		   ((long)tSigScalVar->Y2*tSigScalVar->X1))/
					  		   ((long)tSigScalVar->X2-tSigScalVar->X1));

		/* y zwischen y1 und y2 begrenzen 		*/
		tSigScalVar->Y_SCAL = (short)vxSigBet(vxSigMin(tSigScalVar->Y1,tSigScalVar->Y2),slZwischen,vxSigMax(tSigScalVar->Y1,tSigScalVar->Y2));
	}
	else
	{
		tSigScalVar->ERROR  = 1;
		tSigScalVar->Y_SCAL = 0;
	}
	tSigScalVar->RUN = 0;
}

/**************************************************************/

void xSigScal_R(xSigScal_R_typ *tSigScalVar)
{
	float	slZwischen;

	tSigScalVar->RUN = 1;
	if (tSigScalVar->X2 != tSigScalVar->X1)
	{
		tSigScalVar->ERROR  = 0;

	    /*----------------------------------------------------------*
    	* Berechnung der Skalierung                                 *
	    * Ableitung:    y = k * x + d                               *
    	*                                                           *
	    *               k = (y2-y1) / (x2-x1)                       *
    	*               d = (y1*x2 - y2*x1) / (x2-x1)               *
	    *           ==> y = (x*(y2-y1) + y1*x2 - y2*x1) / (x2-x1)   *
    	*-----------------------------------------------------------*/
    	/* Typkonvertierung auf 32Bit durchführen					*/

		slZwischen = (( (float)(tSigScalVar->X * (tSigScalVar->Y2-tSigScalVar->Y1) +
					  		   (tSigScalVar->Y1*tSigScalVar->X2) -
					  		   (tSigScalVar->Y2*tSigScalVar->X1)) )/
					  		   (float)(tSigScalVar->X2-tSigScalVar->X1));

		/* y zwischen y1 und y2 begrenzen 		*/
		tSigScalVar->Y_SCAL = vxSigBet(vxSigMin(tSigScalVar->Y1,tSigScalVar->Y2),slZwischen,vxSigMax(tSigScalVar->Y1,tSigScalVar->Y2));
	}
	else
	{
		tSigScalVar->ERROR  = 1;
		tSigScalVar->Y_SCAL = 0;
	}
	tSigScalVar->RUN = 0;
}

/**************************************************************
*
*  Zweck:  Schrittregler
*
*  Aufruf: xPISchr(xPISchr_typ *tPISchrVar)
*
*  Übergabep.:    xPISchr_typ-Variable:
*
*  Rückgabep.:
*
*  Beschreibung:
*
*  Datum/Autor:
*  V0.1   08-10-98,BrunnerK   erstellt
*  V0.2   18-07-00,BrunnerK	  Parameter geaendert (AS V1.4 - LibManager)
*
**************************************************************/

void xPISchr(xPISchr_typ *tPISchrVar)
{
	long slXWk;

	if (tPISchrVar->bPIDinit == 0)
	{
		slXWk                = (long)(tPISchrVar->ssX - tPISchrVar->ssW);
		tPISchrVar->slA_XWka = slXWk;
		tPISchrVar->ssdY     =
		    (short)(tPISchrVar->slK * ((slXWk - tPISchrVar->slXWka) +
		    (tPISchrVar->slTI * slXWk)/1000) / 1000 );
	}
	else
	{
		tPISchrVar->ssdY      = 0;
	}
}

/**************************************************************

**************************************************************

**************************************************************/

void xPISchr_R(xPISchr_R_typ *tPISchrVar)
{
	long slXWk;

	if (tPISchrVar->bPIDinit == 0)
	{
		slXWk                = (tPISchrVar->ssX - tPISchrVar->ssW);
		tPISchrVar->slA_XWka = slXWk;
		tPISchrVar->ssdY     =
		    (tPISchrVar->slK * ((slXWk - tPISchrVar->slXWka) +
		    (tPISchrVar->slTI * slXWk)/1000) / 1000 );
	}
	else
	{
		tPISchrVar->ssdY      = 0;
	}
}
```

### Library Logical/Libraries/UniAna_in (IEC, version 0.70.0) - LEGACY CODE- DO NOT USE IN NEW IMPLEMENTATIONS!
